Yaskawa INFORM job: X2_101(P)NEWKM.JBI

/JOB
//NAME X2_101(P)NEWKM
//POS
///NPOS 465,465,465,24,0,0
///TOOL 0
///POSTYPE PULSE
///PULSE
C00000=3858,45070,-46943,-23358,97175,-79306
C00001=-126163,171030,121698,-25332,17066,-72423
///LIMIT ON
C00002=-15532,205449,169164,0,-1122,-37
C00003=-2035,205524,169313,0,-1142,-38
///LIMIT OFF
C00004=-24876,216658,221537,-34735,41227,28422
C00005=-32534,213651,221430,-43713,46730,30831
C00006=-90550,189136,203825,-30202,58765,18284
C00007=-119585,140470,218769,-27614,53519,-2911
C00008=-120519,138494,231532,-24554,52332,-6677
C00009=-121361,123084,224135,-22504,53325,-9347
C00010=-121726,115435,217146,-22627,53645,-9461
C00011=-121876,112275,214159,-22659,53833,-9521
C00012=-121870,108701,209945,-22450,54535,-9681
C00013=-121878,109205,210521,-22481,54446,-9661
C00014=-121910,109175,212145,-22779,53504,-9448
C00015=-121878,109205,210521,-22481,54446,-9661
C00016=-121362,120230,220888,-22358,53819,-9461
C00017=-121399,123144,224213,26030,40987,26163
C00018=-121766,115498,217228,25645,41349,26232
C00019=-121913,110359,211916,25262,41930,26397
C00020=-121910,108768,210034,25105,42240,26494
C00021=-121911,109318,210663,25153,42145,26465
C00022=-121945,109286,212284,25618,41227,26168
C00023=-121911,109318,210663,25153,42145,26465
C00024=-121395,120334,221016,25773,41460,26319
C00025=-121834,122785,223550,29969,46824,26161
C00026=-121859,115436,217233,29902,46923,26193
C00027=-121866,110818,212669,29698,47304,26325
C00028=-121863,108844,210335,29512,47673,26452
C00029=-121935,109447,211025,29521,47579,26410
C00030=-121969,109405,212635,29961,46698,26100
C00031=-121935,109447,211025,29521,47579,26410
C00032=-121897,120013,220389,29693,47285,26314
C00033=-121710,149750,244683,33916,46787,25442
C00034=-122130,167084,227684,35838,62010,28886
C00035=-121679,161325,224182,36290,61247,28722
C00036=-121494,157054,220841,36419,61089,28713
C00037=-121492,155796,219623,36386,61172,28744
C00038=-121498,156274,220057,36390,61156,28737
C00039=-121513,157313,222807,36761,60220,28378
C00040=-121498,156274,220057,36390,61156,28737
C00041=-122131,164491,225278,35793,62131,28930
C00042=-121153,166943,227356,19598,60055,30811
C00043=-121390,161131,223816,19656,59323,30620
C00044=-121486,157179,220857,19658,59138,30564
C00045=-121483,155572,219231,19626,59303,30596
C00046=-121495,156085,219721,19629,59269,30586
C00047=-121510,157133,222481,19854,58176,30378
C00048=-121495,156085,219721,19629,59269,30586
C00049=-121161,164380,224998,19569,60183,30833
C00050=-134270,166899,227330,-30052,67117,-21044
C00051=-134672,161022,223642,-30400,66383,-20931
C00052=-134827,157380,220874,-30511,66205,-20916
C00053=-134816,155436,218995,-30471,66344,-20953
C00054=-134842,155930,219452,-30490,66315,-20951
C00055=-135058,156963,222167,-30845,65285,-20702
C00056=-134842,155930,219452,-30490,66315,-20951
C00057=-134278,164319,224942,-30027,67241,-21080
C00058=-134522,188621,240209,-29351,55882,-39556
C00059=-134281,187845,227413,-27061,47780,-60505
C00060=-134637,183113,225522,-27632,46565,-60252
C00061=-134774,179835,223566,-27858,46107,-60152
C00062=-134763,178280,222255,-27854,46115,-60152
C00063=-134775,178711,222615,-27856,46112,-60156
C00064=-134965,180234,225747,-28400,45052,-59871
C00065=-134775,178711,222615,-27856,46112,-60156
C00066=-134277,185474,225522,-27083,47733,-60488
C00067=-128103,202093,243005,-900,47088,-2105
C00068=-121693,187846,227414,25459,51264,56132
C00069=-121495,183214,225706,25955,50017,55854
C00070=-121414,180043,223882,26152,49543,55743
C00071=-121411,178420,222512,26150,49549,55748
C00072=-121403,178860,222872,26150,49552,55751
C00073=-121416,180408,226053,26590,48508,55442
C00074=-121403,178860,222872,26150,49552,55751
C00075=-121682,185481,225516,25477,51219,56123
C00076=-121689,188183,227953,25513,51119,56094
C00077=-121490,183546,226247,26015,49869,55812
C00078=-121408,180079,224179,26215,49393,55704
C00079=-121407,178755,223064,26213,49397,55705
C00080=-121411,179182,223381,26203,49420,55711
C00081=-121423,180718,226547,26645,48380,55401
C00082=-121411,179182,223381,26203,49420,55711
C00083=-121690,185807,226020,25524,51091,56086
C00084=-123779,190470,236318,58172,45370,-30510
C00085=-122063,184657,229672,57761,45274,-29622
C00086=-121391,180820,225681,57548,45265,-29244
C00087=-121389,179381,224477,57547,45264,-29243
C00088=-121377,179861,224816,57519,45280,-29221
C00089=-121365,178277,221590,56564,45934,-28599
C00090=-121377,179861,224816,57519,45280,-29221
C00091=-121233,179889,223673,56966,45622,-28813
C00092=-120840,179898,223685,57074,45455,-28743
C00093=-121856,179870,223641,56791,45888,-28921
C00094=-124230,188212,233297,57460,45939,-30216
C00095=-135456,214682,237929,8760,44354,-9002
C00096=-135014,207234,230989,8630,44755,-8792
C00097=-134830,202547,226948,8592,44816,-8716
C00098=-134825,201671,226346,8603,44738,-8721
C00099=-134842,202253,226813,8604,44750,-8727
C00100=-134670,200231,223307,8417,45842,-8557
C00101=-134842,202253,226813,8604,44750,-8727
C00102=-135456,212819,236850,8805,44063,-9030
C00103=-144745,210021,243410,8185,41273,-14023
C00104=-162917,179999,233290,6575,38143,-23957
C00105=-161998,172707,226275,6517,38664,-23607
C00106=-162887,167099,219775,6342,39818,-23812
C00107=-162887,165781,218634,6340,39844,-23811
C00108=-162887,166055,218871,6340,39839,-23811
C00109=-162343,164612,215992,6206,40837,-23555
C00110=-162887,166055,218871,6340,39839,-23811
C00111=-162962,177992,231819,6593,38021,-23983
C00112=-147831,180663,236712,-46705,20975,10626
C00113=-148148,173122,227595,-43517,22125,9005
C00114=-148274,168937,222870,-42234,22650,8350
C00115=-148281,167110,221344,-42230,22650,8346
C00116=-148302,167857,221980,-42238,22637,8344
C00117=-147925,166248,218822,-40599,23599,7656
C00118=-148302,167857,221980,-42238,22637,8344
C00119=-147863,178628,235160,-46872,20902,10696
C00120=-134462,161839,227541,-33778,50638,-10353
C00121=-128292,130528,217892,-31335,63768,-21724
C00122=-129684,119449,220047,-34318,57761,-20007
C00123=-130320,112373,214177,-34735,57677,-20053
C00124=-130456,109465,211770,-34840,57652,-20062
C00125=-133214,109388,211257,-36497,57589,-20371
C00126=-136667,109271,210511,-38562,57521,-20784
C00127=-139224,109161,209855,-40060,57485,-21111
C00128=-138850,112080,212320,-39829,57519,-21074
C00129=-138002,119182,218308,-39302,57595,-20992
C00130=-116829,118715,218073,25020,47867,39145
C00131=-117081,112091,213071,24998,47591,39033
C00132=-116945,109370,210997,25124,47467,39017
C00133=-125403,109328,210939,20229,48081,38115
C00134=-125748,112035,212901,19975,48276,38114
C00135=-125224,118667,217955,20186,48522,38233
C00136=-124121,120753,219622,35413,60229,26204
C00137=-123486,114299,214861,35950,59841,26140
C00138=-122342,111487,212696,36731,59624,26198
C00139=-123646,102227,205116,46204,63991,23691
C00140=-125197,104926,207303,45145,64225,23601
C00141=-126541,111461,212474,44185,64527,23570
C00142=-123354,156374,234537,36141,60524,36841
C00143=-123006,163587,222304,33363,70023,40058
C00144=-122562,159556,221336,33872,68682,39742
C00145=-122328,157903,220938,34117,68123,39618
C00146=-120667,157882,220896,34940,67759,39903
C00147=-118950,157779,220838,35793,67346,40185
C00148=-123086,151768,218649,44650,69367,37665
C00149=-123645,153585,219325,44221,69895,37762
C00150=-124560,157673,220588,43425,71117,38069
C00151=-118179,162280,221931,19519,66647,42953
C00152=-118374,158121,220823,19639,65298,42675
C00153=-118267,155527,219476,19766,64809,42612
C00154=-124138,155466,219359,17061,65585,41471
C00155=-124017,158021,220644,17053,66071,41570
C00156=-123705,162202,221801,17023,67409,41838
C00157=-131226,163758,224551,-30632,74582,-25473
C00158=-131671,158900,222412,-31029,73469,-25265
C00159=-131767,156865,221384,-31140,73093,-25182
C00160=-137554,155593,218490,-34050,72807,-26431
C00161=-137282,157641,219617,-33852,73169,-26479
C00162=-136745,162505,221837,-33401,74244,-26683
C00163=-132458,177728,230704,-28826,51363,-58996
C00164=-131589,185090,225420,-26277,57937,-60697
C00165=-131989,181524,225146,-26843,56352,-60401
C00166=-132129,179690,224573,-27052,55792,-60292
C00167=-137018,178141,221655,-27936,55567,-61763
C00168=-136911,179846,222046,-27715,56157,-61897
C00169=-136440,196977,232068,-26852,58624,-62420
C00170=-123981,183157,222393,21512,66418,58052
C00171=-123825,180405,223212,21872,64600,57740
C00172=-123515,178835,223292,22117,63748,57656
C00173=-118554,178759,223273,23717,62772,58838
C00174=-118823,180539,223431,23475,63574,58935
C00175=-119074,183322,222662,23052,65379,59248
C00176=-122702,184077,222510,27150,66928,58165
C00177=-122303,181421,223407,27656,65122,57824
C00178=-121939,179837,223488,27962,64268,57706
C00179=-119147,179825,223466,28889,63614,58349
C00180=-122880,176137,223692,38896,64069,56161
C00181=-123433,177900,223899,38463,64850,56297
C00182=-124245,180658,223301,37680,66520,56676
C00183=-126373,202040,241637,26852,43466,21020
C00184=-128666,178893,235276,24840,16714,-14065
C00185=-128229,171381,226060,22241,18307,-12727
C00186=-128063,167759,221784,21279,19001,-12231
C00187=-126454,168065,222273,20329,18606,-11329
C00188=-113498,168020,221950,9782,17256,-2783
C00189=-116924,165235,218756,37372,21894,-17093
C00190=-117333,168644,222995,38850,21324,-17919
C00191=-117978,176136,232334,42331,20047,-19764
C00192=-122460,189534,236128,2418,24460,-9718
C00193=-126271,180528,223816,-31550,27550,-1309
C00194=-126367,172058,213874,-29849,29054,-2198
C00195=-127090,167664,208219,-28567,29945,-3048
C00196=-142506,160672,196064,-19689,30087,-11601
C00197=-142606,164949,201311,-20262,29094,-11331
C00198=-142831,174249,212461,-21540,27099,-10741
C00199=-90550,189136,203825,-30202,58765,18284
C00200=-32534,213651,221430,-43713,46730,30831
///LIMIT ON
C00201=-2035,205524,169313,0,-1142,-38
///LIMIT OFF
C00202=110357,194361,192639,11084,17793,24068
C00203=114624,170501,213981,27000,30394,20280
C00204=117760,152303,229663,38696,39653,17494
C00205=136745,136971,237540,47053,40245,16937
C00206=147677,120644,222935,49307,45765,18910
C00207=147943,109722,211385,48401,46737,19631
C00208=147915,107740,209041,48089,47029,19824
C00209=147921,108247,209621,48160,46963,19780
C00210=148534,108214,211137,49208,46239,19387
C00211=147921,108247,209621,48160,46963,19780
C00212=146752,119366,220398,48075,46495,19266
C00213=146769,122228,223642,-12245,42312,-23405
C00214=147600,114525,216379,-11673,42843,-23379
C00215=143912,110143,217361,-5106,40312,-21729
C00216=143912,106051,212649,-5023,41107,-21780
C00217=143912,106490,213159,-5032,41020,-21775
C00218=144459,106367,214517,-4806,40132,-21665
C00219=143912,108428,215397,-5071,40640,-21751
C00220=146723,119408,220432,-12150,42825,-23484
C00221=143045,138896,235476,-13742,43230,-24222
C00222=120960,164034,232760,-20897,55487,-30119
C00223=121057,160229,229930,-20909,55300,-30059
C00224=121055,158546,228333,-20881,55408,-30082
C00225=121067,159042,228799,-20882,55381,-30074
C00226=121067,159823,231250,-21156,54345,-29857
C00227=121067,159042,228799,-20882,55381,-30074
C00228=120732,167440,234058,-20772,56349,-30345
C00229=148415,169733,235789,37593,61151,22296
C00230=149007,163695,231894,38120,60456,22164
C00231=149231,159863,228946,38284,60282,22149
C00232=149211,158151,227325,38234,60380,22184
C00233=149239,158627,227750,38254,60361,22183
C00234=149676,159369,230053,38836,59445,21914
C00235=149239,158627,227750,38254,60361,22183
C00236=148408,167213,233502,37553,61243,22331
C00237=120948,174757,250553,37714,32624,49250
C00238=118901,165188,232218,31966,38533,51583
C00239=120946,159930,222884,30547,40745,53182
C00240=121038,156296,220141,30673,40571,53142
C00241=121036,154340,218237,30574,40715,53200
C00242=121048,154616,218515,30593,40687,53192
C00243=121049,155465,220596,31099,39958,52886
C00244=121048,154822,218707,30600,40677,53188
C00245=120729,163160,224069,29968,41598,53447
C00246=121377,165750,226457,-30289,41550,-53313
C00247=121143,159913,222862,-30795,40818,-53099
C00248=121047,156279,220118,-30922,40645,-53059
C00249=121045,154323,218215,-30823,40788,-53119
C00250=121036,154817,218686,-30845,40755,-53109
C00251=121036,155874,221461,-31554,39751,-52691
C00252=121036,154817,218686,-30845,40755,-53109
C00253=121366,163152,224045,-30207,41677,-53367
C00254=121366,163152,224045,-30207,41677,-53367
C00255=121483,199612,234227,-6189,47888,801
C00256=116205,204502,245408,11942,36344,-5913
C00257=116205,198287,241356,12142,35658,-6024
C00258=115285,196386,239785,12255,35742,-6372
C00259=115285,194113,238215,12313,35542,-6405
C00260=115285,196386,239785,12255,35742,-6372
C00261=115348,194991,237157,11988,36617,-6206
C00262=115285,196386,239785,12255,35742,-6372
C00263=123104,195479,239507,19665,35466,-6181
C00264=123104,195479,239507,19665,35466,-6181
C00265=123104,193192,237914,19758,35282,-6230
C00266=123104,195479,239507,19665,35466,-6181
C00267=123076,194119,236930,19261,36311,-5967
C00268=123104,195479,239507,19665,35466,-6181
C00269=121128,212741,249815,-1743,43167,1820
C00270=122107,209686,246756,-2334,35321,2429
C00271=122102,206275,244139,-2341,35179,2433
C00272=122102,203894,242650,-2356,34872,2441
C00273=122102,204632,243115,-2351,34965,2438
C00274=122089,203132,240589,-2306,35750,2407
C00275=122102,206496,244275,-2336,35209,2431
C00276=106576,204382,240236,-11557,35635,-12
C00277=105844,202338,238595,-11416,35522,-303
C00278=105844,200288,237272,-11482,35287,-265
C00279=105844,200808,237609,-11466,35345,-274
C00280=105986,199498,235274,-11288,36108,-332
C00281=106675,205315,241966,-11744,35073,120
C00282=121297,207453,245813,-14870,35545,6164
C00283=121834,203391,244226,-16112,31944,7027
C00284=106221,199743,239162,-19916,31296,2840
C00285=113509,210579,250034,-22345,31553,6212
C00286=137477,186722,245503,32144,20066,-8132
C00287=144465,175669,236908,30012,18300,-5031
C00288=139549,172315,235287,31351,18759,-7203
C00289=137345,164078,227518,10851,18120,-89
C00290=146058,157132,216606,32577,20921,-6799
C00291=140284,173520,236299,40392,19304,-12229
C00292=141359,173291,233520,11184,20569,1731
C00293=118409,183246,223281,22704,61297,57282
C00294=118581,179790,223172,23116,59682,56982
C00295=119080,177311,221631,23320,59284,57040
C00296=121941,178499,224734,27845,56338,58798
C00297=123595,179764,223148,24469,58676,58234
C00298=123340,183247,223305,24003,60279,58531
C00299=123969,187046,227095,-21794,65540,-58072
C00300=123769,179484,222767,-22062,64364,-57894
C00301=123576,177800,222588,-22257,63628,-57801
C00302=118799,177973,222710,-23788,62722,-58944
C00303=118761,179531,222831,-23662,63378,-59098
C00304=119022,182337,222102,-23232,65173,-59409
C00305=118548,185960,240006,-23112,60518,-52609
C00306=118308,157164,220237,-19921,65161,-42814
C00307=118476,159354,225951,-20677,60172,-41891
C00308=123703,159378,225931,-18342,60853,-40897
C00309=124532,167340,231429,-17858,61624,-40849
C00310=131317,177717,239716,826,64580,-18015
C00311=127714,174798,240675,21893,68906,13109
C00312=128493,175754,243778,32993,66237,18094
C00313=129602,162263,233964,31751,67819,21399
C00314=133248,162950,235869,37514,65238,22588
C00315=131009,170167,241494,36207,65881,22354
C00316=129314,152311,241224,32836,60701,20495
C00317=134262,125348,219975,36015,59621,20953
C00318=135447,125082,223354,38338,54808,19572
C00319=142546,124299,220540,42255,55214,20638
C00320=139661,130867,226583,40618,55342,20260
C00321=128999,132996,229263,10730,53492,-5640
C00322=116671,118195,219736,-25901,46707,-38928
C00323=118115,111302,212748,-24760,47506,-38978
C00324=115332,106344,206919,-23218,48620,-39011
C00325=123639,106372,207077,-18510,49117,-38052
C00326=123644,119783,222350,-19919,44975,-37125
C00327=114229,133215,224760,-34569,55636,-15897
C00328=115215,137513,213650,-31198,63454,-18326
C00329=115698,129470,194907,-29425,69976,-20075
C00330=106762,152299,200628,-28970,57173,-24551
C00331=110317,154116,190151,-51141,5677,-13903
C00332=107071,171086,183471,-26129,-3539,-25752
C00333=106762,173596,155880,-23749,-4416,-26879
C00334=27327,173596,155880,-23749,-4416,-26879
C00335=61821,209309,227101,13653,32656,17858
C00336=117760,152303,229663,38696,39653,17494
C00337=136745,136971,237540,47053,40245,16937
C00338=146994,113665,215692,48512,45897,19228
C00339=147943,109722,211385,48401,46737,19631
C00340=147915,107740,209041,48089,47029,19824
C00341=147921,108247,209621,48160,46963,19780
C00342=148534,108214,211137,49208,46239,19387
C00343=147921,108247,209621,48160,46963,19780
C00344=146752,119366,220398,48075,46495,19266
C00345=146769,122228,223642,-12245,42312,-23405
C00346=147600,114525,216379,-11673,42843,-23379
C00347=150410,110151,217690,-10757,39930,-22674
C00348=147891,107738,209025,-11299,43871,-23478
C00349=153573,108674,222079,-9620,36586,-21959
C00350=148504,108258,211178,-11182,42854,-23269
C00351=153573,108674,222079,-9620,36586,-21959
C00352=146723,119408,220432,-12150,42825,-23484
C00353=145733,131948,231566,-12791,42388,-23541
C00354=120722,165761,226456,-19970,59936,-31049
C00355=120948,159926,222866,-20032,59223,-30862
C00356=121040,156088,219926,-20029,59083,-30814
C00357=121038,154338,218222,-19999,59222,-30841
C00358=121049,154854,218719,-20002,59186,-30831
C00359=121049,155913,221496,-20240,58090,-30621
C00360=121049,154854,218719,-20002,59186,-30831
C00361=120732,163185,224070,-19939,60073,-31072
C00362=147021,165785,226508,35831,64459,23179
C00363=147568,159794,222565,36267,63796,23080
C00364=147776,155921,219507,36395,63658,23083
C00365=147758,154144,217781,36345,63784,23124
C00366=147784,154635,218233,36365,63757,23122
C00367=148179,155632,220846,36870,62776,22859
C00368=147784,154635,218233,36365,63757,23122
C00369=147016,163193,224095,35787,64586,23223
C00370=120935,171934,242189,34504,35645,50983
C00371=120720,165768,226479,30046,41476,53396
C00372=120946,159930,222884,30547,40745,53182
C00373=121038,156296,220141,30673,40571,53142
C00374=121036,154340,218237,30574,40715,53200
C00375=121048,154616,218515,30593,40687,53192
C00376=121049,155465,220596,31099,39958,52886
C00377=121048,154822,218707,30600,40677,53188
C00378=120729,163160,224069,29968,41598,53447
C00379=121377,165750,226457,-30289,41550,-53313
C00380=121143,159913,222862,-30795,40818,-53099
C00381=121047,156279,220118,-30922,40645,-53059
C00382=121045,154323,218215,-30823,40788,-53119
C00383=121036,154817,218686,-30845,40755,-53109
C00384=121036,155874,221461,-31554,39751,-52691
C00385=121036,154817,218686,-30845,40755,-53109
C00386=121366,163152,224045,-30207,41677,-53367
C00387=137298,197580,228407,-4602,50872,8306
C00388=150104,186063,215083,4172,47395,10089
C00389=151037,187915,222611,5560,37459,9696
C00390=151037,185231,220636,5579,37292,9686
C00391=151037,186381,221487,5571,37359,9691
C00392=150722,184726,218590,5524,38303,9628
C00393=151037,186381,221487,5571,37359,9691
C00394=146916,195279,232433,6810,35442,7817
C00395=137844,201998,246759,9498,27003,3396
C00396=137686,197394,242433,9461,27307,3368
C00397=137686,195263,240973,9523,27113,3337
C00398=137686,196472,241804,9489,27221,3355
C00399=137493,195182,239322,9290,28089,3401
C00400=137686,196472,241804,9489,27221,3355
C00401=137872,200789,246191,9576,26732,3366
C00402=125774,205155,244676,-1779,39656,5291
C00403=112923,203838,248508,-13462,25066,7526
C00404=112273,198134,243408,-13075,25198,7148
C00405=112273,195800,241814,-13181,24982,7201
C00406=112273,196433,242252,-13153,25040,7187
C00407=112372,195114,239703,-12779,25919,7028
C00408=112273,198506,243659,-13056,25235,7140
C00409=116013,198964,244548,-14816,25354,9073
C00410=116342,198570,244149,-14930,25435,9223
C00411=116342,196143,242500,-15057,25209,9285
C00412=116342,196705,242885,-15029,25259,9270
C00413=116387,195582,240705,-14639,26004,9089
C00414=116342,197910,243703,-14967,25370,9239
C00415=117942,195646,241316,-14532,25786,9480
C00416=100647,189294,231884,-21448,26183,5644
C00417=105174,198018,242573,-25014,25112,8670
C00418=138600,188940,247456,26519,19021,-5159
C00419=137571,174455,238189,28708,17651,-6518
C00420=137161,164520,226883,26329,19378,-5524
C00421=155042,153638,205005,15246,25339,2538
C00422=152712,160990,215450,17982,23102,538
C00423=143867,184578,245341,28376,18738,-7025
C00424=118409,183246,223281,22704,61297,57282
C00425=118581,179790,223172,23116,59682,56982
C00426=118693,177304,221659,23221,59339,56941
C00427=123485,177367,221685,24518,58397,58134
C00428=123595,179764,223148,24469,58676,58234
C00429=123340,183247,223305,24003,60279,58531
C00430=123938,190075,227776,-21625,66593,-58285
C00431=123769,179484,222767,-22062,64364,-57894
C00432=123184,178126,222935,-22395,63511,-57887
C00433=118491,177814,222796,-23918,62536,-58992
C00434=118761,179531,222831,-23662,63378,-59098
C00435=119022,182337,222102,-23232,65173,-59409
C00436=122719,191364,242917,-21569,61694,-52463
C00437=118308,157164,220237,-19921,65161,-42814
C00438=118111,154516,218858,-20091,64650,-42768
C00439=123565,154529,218888,-17585,65335,-41706
C00440=123968,157132,220198,-17330,65894,-41703
C00441=123666,171172,229916,-17315,67038,-41943
C00442=144355,163571,225284,37353,71372,27423
C00443=145029,158578,222871,37922,70344,27214
C00444=145301,156779,221933,38139,70000,27151
C00445=150377,154595,216968,40372,70234,28530
C00446=150395,156248,217650,40288,70560,28668
C00447=149652,161243,220185,39700,71542,28858
C00448=132795,148549,237387,35039,60818,21489
C00449=129694,120788,221943,34103,57517,19821
C00450=131382,111553,213551,35044,57698,20084
C00451=141801,108057,208206,41145,57678,21431
C00452=149498,107271,204816,45301,57831,22696
C00453=138916,111308,211941,39557,57554,20977
C00454=138073,118434,217968,39036,57618,20892
C00455=116671,118195,219736,-25901,46707,-38928
C00456=118115,111302,212748,-24760,47506,-38978
C00457=116900,108123,210017,-25446,47458,-39118
C00458=125154,108371,210177,-20660,48073,-38243
C00459=125733,111262,212625,-20332,48091,-38177
C00460=125221,117920,217723,-20539,48325,-38292
C00461=126776,138177,229575,-26069,55844,-18031
C00462=78165,188060,235135,7900,30611,9082
C00463=59194,210722,234815,16854,29215,15555
C00464=-5072,204191,177105,2520,2910,2072
BC00000=46343,515539,1075137
BC00001=134211,257442,1075137
BC00002=1577,514581,1075193
///LIMIT ON
BC00003=1577,-59411,1075193
BC00004=21651,-83121,1075193
BC00005=24420,-86391,1075193
BC00006=182796,-159531,881707
BC00007=261191,-81513,996983
BC00008=265032,-63260,961437
BC00009=267226,-52830,941125
BC00010=267226,-52830,941125
BC00011=267226,-52830,941125
BC00012=267226,-52830,941125
BC00013=267226,-52830,941125
BC00014=267226,-52830,941125
BC00015=267226,-52830,941125
BC00016=267226,-52830,941125
BC00017=280671,-69653,979309
BC00018=280671,-69653,979309
BC00019=280671,-69653,979309
BC00020=280671,-69653,979309
BC00021=280671,-69653,979309
BC00022=280671,-69653,979309
BC00023=280671,-69653,979309
BC00024=280671,-69653,979309
BC00025=340059,-63189,958778
BC00026=340059,-63189,958778
BC00027=340059,-63189,958778
BC00028=340059,-63189,958778
BC00029=340059,-63189,958778
BC00030=340059,-63189,958778
BC00031=340059,-63189,958778
BC00032=340059,-63189,958778
BC00033=335398,-76723,919166
BC00034=322582,-113941,810232
BC00035=322582,-113941,810232
BC00036=322582,-113941,810232
BC00037=322582,-113941,810232
BC00038=322582,-113941,810232
BC00039=322582,-113941,810232
BC00040=322582,-113941,810232
BC00041=322582,-113941,810232
BC00042=280667,-107560,836160
BC00043=280667,-107560,836160
BC00044=280667,-107560,836160
BC00045=280667,-107560,836160
BC00046=280667,-107560,836160
BC00047=280667,-107560,836160
BC00048=280667,-107560,836160
BC00049=280667,-107560,836160
BC00050=310567,-93619,803899
BC00051=310567,-93619,803899
BC00052=310567,-93619,803899
BC00053=310567,-93619,803899
BC00054=310567,-93619,803899
BC00055=310567,-93619,803899
BC00056=310567,-93619,803899
BC00057=310567,-93619,803899
BC00058=310965,-106510,799405
BC00059=311390,-120260,794612
BC00060=311390,-120260,794612
BC00061=311390,-120260,794612
BC00062=311390,-120260,794612
BC00063=311390,-120260,794612
BC00064=311390,-120260,794612
BC00065=311390,-120260,794612
BC00066=311390,-120260,794612
BC00067=292086,-121797,794251
BC00068=272781,-123335,793890
BC00069=272781,-123335,793890
BC00070=272781,-123335,793889
BC00071=272781,-123335,793890
BC00072=272781,-123335,793890
BC00073=272781,-123335,793890
BC00074=272781,-123335,793890
BC00075=272781,-123335,793890
BC00076=341329,-123426,794084
BC00077=341329,-123426,794084
BC00078=341329,-123426,794084
BC00079=341329,-123426,794084
BC00080=341329,-123426,794084
BC00081=341329,-123426,794084
BC00082=341329,-123426,794084
BC00083=341329,-123426,794084
BC00084=311173,-145946,723752
BC00085=311173,-145946,723752
BC00086=311173,-145946,723752
BC00087=311173,-145946,723752
BC00088=311173,-145946,723752
BC00089=311173,-145946,723752
BC00090=311173,-145946,723752
BC00091=311173,-145946,723752
BC00092=311173,-145946,723752
BC00093=311173,-145946,723752
BC00094=311173,-145946,723752
BC00095=368417,-159833,659013
BC00096=368417,-159833,659013
BC00097=368417,-159833,659013
BC00098=368417,-159833,659013
BC00099=368417,-159833,659013
BC00100=368417,-159833,659013
BC00101=368417,-159833,659013
BC00102=368417,-159833,659013
BC00103=371175,-130977,746316
BC00104=376801,-72111,924416
BC00105=376801,-72111,924416
BC00106=376801,-72111,924416
BC00107=376801,-72111,924416
BC00108=376801,-72111,924416
BC00109=376801,-72111,924414
BC00110=376801,-72111,924416
BC00111=376801,-72111,924416
BC00112=341502,-110623,881707
BC00113=341502,-110623,881707
BC00114=341502,-110623,881707
BC00115=341502,-110623,881707
BC00116=341502,-110623,881707
BC00117=341502,-110623,881707
BC00118=341502,-110623,881707
BC00119=341502,-110623,881707
BC00120=317229,-102231,901443
BC00121=301231,-72103,952987
BC00122=300570,-48582,912240
BC00123=300570,-48582,912240
BC00124=300570,-48582,912238
BC00125=300570,-48582,912240
BC00126=300570,-48582,912240
BC00127=300570,-48582,912240
BC00128=300570,-48582,912240
BC00129=300570,-48582,912240
BC00130=280392,-58723,951442
BC00131=280392,-58723,951442
BC00132=280392,-58723,951442
BC00133=280392,-58723,951442
BC00134=280392,-58723,951442
BC00135=280392,-58723,951442
BC00136=316381,-56573,892692
BC00137=316381,-56573,892692
BC00138=316381,-56573,892692
BC00139=316381,-56573,892692
BC00140=316381,-56573,892692
BC00141=316381,-56573,892692
BC00142=316378,-102850,892874
BC00143=316296,-103943,772800
BC00144=316296,-103943,772800
BC00145=316296,-103943,772800
BC00146=316296,-103943,772800
BC00147=316296,-103943,772800
BC00148=316296,-103943,772800
BC00149=316296,-103943,772800
BC00150=316296,-103943,772800
BC00151=280455,-96630,809993
BC00152=280455,-96630,809993
BC00153=280455,-96630,809993
BC00154=280455,-96630,809993
BC00155=280455,-96630,809993
BC00156=280455,-96630,809993
BC00157=313485,-85360,768647
BC00158=313485,-85360,768647
BC00159=313485,-85360,768647
BC00160=313485,-85360,768647
BC00161=313485,-85360,768647
BC00162=313485,-85360,768647
BC00163=312825,-103474,920081
BC00164=312211,-104211,778577
BC00165=312211,-104211,778577
BC00166=312212,-104211,778575
BC00167=312212,-104211,778575
BC00168=312211,-104211,778577
BC00169=312211,-104211,778577
BC00170=271148,-98769,766614
BC00171=271148,-98769,766614
BC00172=271148,-98769,766614
BC00173=271148,-98769,766614
BC00174=271148,-98769,766614
BC00175=271148,-98769,766614
BC00176=325606,-102154,751502
BC00177=325606,-102154,751502
BC00178=325606,-102154,751502
BC00179=325606,-102154,751502
BC00180=325606,-102154,751502
BC00181=325606,-102154,751502
BC00182=325606,-102154,751502
BC00183=333034,-134164,767871
BC00184=339129,-149656,848222
BC00185=339129,-149656,848222
BC00186=339128,-149655,848221
BC00187=339129,-149656,848222
BC00188=339129,-149656,848222
BC00189=339129,-149656,848222
BC00190=339129,-149656,848222
BC00191=339129,-149656,848222
BC00192=327972,-150195,844855
BC00193=317352,-148908,839217
BC00194=317352,-148908,839217
BC00195=317352,-148908,839217
BC00196=317352,-148908,839217
BC00197=317352,-148908,839217
BC00198=317352,-148908,839217
BC00199=182796,-159531,881707
BC00200=24420,-86391,1075193
BC00201=1577,-59411,1075193
///LIMIT OFF
BC00202=66886,568997,1042628
BC00203=92444,428784,1010343
BC00204=92897,349346,986620
BC00205=164885,323227,963040
BC00206=185515,310988,951990
BC00207=185515,310988,951990
BC00208=185515,310988,951990
BC00209=185515,310988,951990
BC00210=185515,310988,951990
BC00211=185515,310988,951990
BC00212=185515,310988,951990
BC00213=189482,318421,980677
BC00214=189482,318421,980677
BC00215=189482,306857,980677
BC00216=189482,306857,980677
BC00217=189482,306857,980677
BC00218=189482,306857,980677
BC00219=189482,306857,980677
BC00220=189482,318421,980677
BC00221=182754,323413,960497
BC00222=141913,353717,838001
BC00223=141913,353717,838001
BC00224=141913,353717,838001
BC00225=141913,353717,838001
BC00226=141913,353717,838001
BC00227=141913,353717,838001
BC00228=141913,353717,838001
BC00229=207263,329283,804361
BC00230=207263,329283,804361
BC00231=207263,329283,804361
BC00232=207263,329283,804361
BC00233=207263,329283,804361
BC00234=207263,329283,804361
BC00235=207263,329283,804361
BC00236=207263,329283,804361
BC00237=131545,342192,928572
BC00238=131545,342192,928572
BC00239=131545,352945,928572
BC00240=131545,352945,928572
BC00241=131545,352945,928572
BC00242=131545,352945,928572
BC00243=131546,352945,928571
BC00244=131545,352945,928572
BC00245=131545,352945,928572
BC00246=134650,353410,929381
BC00247=134650,353410,929381
BC00248=134650,353410,929381
BC00249=134650,353410,929381
BC00250=134650,353410,929381
BC00251=134650,353410,929381
BC00252=134650,353410,929381
BC00253=134650,353410,929381
BC00254=134650,353410,929381
BC00255=134373,390505,753296
BC00256=93548,390505,753296
BC00257=93548,390505,753296
BC00258=93548,390505,753296
BC00259=93548,390505,753296
BC00260=93548,390505,753296
BC00261=93548,390505,753296
BC00262=93548,390505,753296
BC00263=93548,390505,753296
BC00264=93548,390505,753296
BC00265=93548,390505,753296
BC00266=93548,390505,753296
BC00267=93548,390505,753296
BC00268=93548,390505,753296
BC00269=168621,382981,746953
BC00270=168621,382981,746953
BC00271=168621,382981,746953
BC00272=168621,382981,746953
BC00273=168621,382981,746953
BC00274=168621,382981,746953
BC00275=168621,382981,746953
BC00276=147987,382981,746953
BC00277=147987,382981,746953
BC00278=147987,382981,746953
BC00279=147987,382981,746953
BC00280=147987,382981,746953
BC00281=147987,382981,746953
BC00282=147987,382981,746953
BC00283=148413,382917,748107
BC00284=148720,382872,748941
BC00285=148720,382872,748941
BC00286=202687,374937,895402
BC00287=202687,374937,895402
BC00288=181755,375248,897598
BC00289=159634,375248,897598
BC00290=159830,375278,897817
BC00291=159830,375278,897817
BC00292=181599,378656,922199
BC00293=133265,363347,778304
BC00294=133265,363347,778304
BC00295=133265,363348,778302
BC00296=133265,363347,778303
BC00297=133265,363347,778304
BC00298=133265,363347,778304
BC00299=146867,355192,768709
BC00300=133835,355192,768709
BC00301=133835,355192,768709
BC00302=133835,355192,768709
BC00303=133835,355192,768709
BC00304=133835,355192,768709
BC00305=137056,354441,784011
BC00306=142942,353070,811970
BC00307=142942,353070,811970
BC00308=142942,353070,811970
BC00309=142942,353070,811970
BC00310=165851,345786,796984
BC00311=162229,334955,774700
BC00312=164558,332161,768952
BC00313=169097,331686,770079
BC00314=169097,331686,770079
BC00315=169097,331686,770079
BC00316=172928,318668,849125
BC00317=172716,318424,871943
BC00318=172716,318424,871943
BC00319=172716,318424,871943
BC00320=172716,318424,871943
BC00321=159709,316953,907603
BC00322=143169,315083,952947
BC00323=143169,315083,952947
BC00324=143169,315083,952947
BC00325=143169,315083,952947
BC00326=143169,315083,952947
BC00327=119317,333024,923162
BC00328=123697,333024,923162
BC00329=132263,359008,1050367
BC00330=116798,380944,1050367
BC00331=119098,435388,1050366
BC00332=102300,494697,1050367
BC00333=98226,585882,1050367
BC00334=13715,585882,1050367
BC00335=124194,427082,1056800
BC00336=295181,349346,986620
BC00337=336555,323227,963040
BC00338=354347,311995,952900
BC00339=355943,310988,951990
BC00340=355943,310988,951990
BC00341=355943,310988,951990
BC00342=355943,310988,951990
BC00343=355943,310988,951990
BC00344=355943,310988,951990
BC00345=359910,318421,980677
BC00346=359910,318421,980677
BC00347=359910,306857,980677
BC00348=359910,318421,980677
BC00349=359910,294465,980677
BC00350=359910,318421,980677
BC00351=359910,294465,980677
BC00352=359910,318421,980677
BC00353=359910,318421,980677
BC00354=312341,364470,838001
BC00355=312341,364470,838001
BC00356=312341,364470,838001
BC00357=312341,364470,838001
BC00358=312341,364470,838001
BC00359=312341,364470,838001
BC00360=312341,364470,838001
BC00361=312341,364470,838001
BC00362=377691,340036,804361
BC00363=377691,340036,804361
BC00364=377691,340036,804361
BC00365=377691,340036,804361
BC00366=377691,340036,804361
BC00367=377691,340036,804361
BC00368=377691,340036,804361
BC00369=377691,340036,804361
BC00370=301973,352945,928572
BC00371=301973,352945,928572
BC00372=301973,352945,928572
BC00373=301973,352945,928572
BC00374=301973,352945,928572
BC00375=301973,352945,928572
BC00376=301974,352945,928571
BC00377=301973,352945,928572
BC00378=301973,352945,928572
BC00379=305078,353410,929381
BC00380=305078,353410,929381
BC00381=305078,353410,929381
BC00382=305078,353410,929381
BC00383=305078,353410,929381
BC00384=305078,353410,929381
BC00385=305078,353410,929381
BC00386=305078,353410,929381
BC00387=355079,392127,745599
BC00388=333047,392127,745599
BC00389=333047,392127,745599
BC00390=333047,392127,745599
BC00391=333047,392127,745599
BC00392=333047,392127,745599
BC00393=333047,392127,745599
BC00394=333047,392127,745599
BC00395=333047,392127,745599
BC00396=333047,392127,745599
BC00397=333047,392127,745599
BC00398=333047,392127,745599
BC00399=333047,392127,745599
BC00400=333047,392127,745599
BC00401=333047,392127,745599
BC00402=330711,385408,779676
BC00403=330711,385408,779676
BC00404=330711,385408,779676
BC00405=330711,385408,779676
BC00406=330711,385408,779676
BC00407=330711,385408,779676
BC00408=330711,385408,779676
BC00409=286508,385408,779676
BC00410=286508,385408,779676
BC00411=286508,385408,779676
BC00412=286508,385408,779676
BC00413=286508,385408,779676
BC00414=286508,385408,779676
BC00415=288154,385206,781872
BC00416=288360,385181,782147
BC00417=288360,385181,782147
BC00418=340469,375654,887477
BC00419=340973,375751,888339
BC00420=340973,375751,888339
BC00421=341056,375767,888482
BC00422=341056,375767,888482
BC00423=341056,375767,888482
BC00424=303693,363347,778304
BC00425=303693,363347,778304
BC00426=303693,363348,778302
BC00427=303693,363347,778303
BC00428=303693,363347,778304
BC00429=303693,363347,778304
BC00430=304263,355192,768709
BC00431=304263,355192,768709
BC00432=304263,355192,768709
BC00433=304263,355192,768709
BC00434=304263,355192,768709
BC00435=304263,355192,768709
BC00436=307126,354525,782310
BC00437=313370,353070,811970
BC00438=313370,353070,811970
BC00439=313370,353070,811970
BC00440=313370,353070,811970
BC00441=313370,353070,811970
BC00442=381578,331383,767352
BC00443=381578,331383,767352
BC00444=381578,331383,767352
BC00445=381578,331383,767352
BC00446=381578,331383,767352
BC00447=381578,331383,767352
BC00448=337601,317122,860141
BC00449=333177,303767,911398
BC00450=333177,303767,911398
BC00451=353932,303767,911398
BC00452=353932,303767,911398
BC00453=333177,303767,911398
BC00454=333177,303767,911398
BC00455=313597,315083,952947
BC00456=313597,315083,952947
BC00457=313597,315083,952947
BC00458=313597,315083,952947
BC00459=313597,315083,952947
BC00460=313597,315083,952947
BC00461=317033,330359,927586
BC00462=204139,405669,1028194
BC00463=121307,427031,1056816
BC00464=21523,502292,1072610
EC00000=-1108551,372643
EC00001=-1108551,372643
EC00002=-1108551,372643
EC00003=-1108551,372643
EC00004=-1108551,372643
EC00005=-1108551,372643
EC00006=-1108551,372643
EC00007=-1108551,372643
EC00008=-1108551,372643
EC00009=-1108551,372643
EC00010=-1108551,372643
EC00011=-1108551,372643
EC00012=-1108551,372643
EC00013=-1108551,372643
EC00014=-1108551,372643
EC00015=-1108551,372643
EC00016=-1108551,372643
EC00017=-1108551,372643
EC00018=-1108551,372643
EC00019=-1108551,372643
EC00020=-1108551,372643
EC00021=-1108551,372643
EC00022=-1108551,372643
EC00023=-1108551,372643
EC00024=-1108551,372643
EC00025=-1108551,372643
EC00026=-1108551,372643
EC00027=-1108551,372643
EC00028=-1108551,372643
EC00029=-1108551,372643
EC00030=-1108551,372643
EC00031=-1108551,372643
EC00032=-1108551,372643
EC00033=-1108551,372643
EC00034=-1108551,372643
EC00035=-1108551,372643
EC00036=-1108551,372643
EC00037=-1108551,372643
EC00038=-1108551,372643
EC00039=-1108551,372643
EC00040=-1108551,372643
EC00041=-1108551,372643
EC00042=-1108551,372643
EC00043=-1108551,372643
EC00044=-1108551,372643
EC00045=-1108551,372643
EC00046=-1108551,372643
EC00047=-1108551,372643
EC00048=-1108551,372643
EC00049=-1108551,372643
EC00050=-1108551,372643
EC00051=-1108551,372643
EC00052=-1108551,372643
EC00053=-1108551,372643
EC00054=-1108551,372643
EC00055=-1108551,372643
EC00056=-1108551,372643
EC00057=-1108551,372643
EC00058=-1108551,372643
EC00059=-1108551,372643
EC00060=-1108551,372643
EC00061=-1108551,372643
EC00062=-1108551,372643
EC00063=-1108551,372643
EC00064=-1108551,372643
EC00065=-1108551,372643
EC00066=-1108551,372643
EC00067=-1108551,372643
EC00068=-1108551,372643
EC00069=-1108551,372643
EC00070=-1108550,372643
EC00071=-1108551,372643
EC00072=-1108551,372643
EC00073=-1108551,372643
EC00074=-1108551,372643
EC00075=-1108551,372643
EC00076=-1108551,372643
EC00077=-1108551,372643
EC00078=-1108551,372643
EC00079=-1108551,372643
EC00080=-1108551,372643
EC00081=-1108551,372643
EC00082=-1108551,372643
EC00083=-1108551,372643
EC00084=-1108551,372643
EC00085=-1108551,372643
EC00086=-1108551,372643
EC00087=-1108551,372643
EC00088=-1108551,372643
EC00089=-1108551,372643
EC00090=-1108551,372643
EC00091=-1108551,372643
EC00092=-1108551,372643
EC00093=-1108551,372643
EC00094=-1108551,372643
EC00095=-1108551,372643
EC00096=-1108551,372643
EC00097=-1108551,372643
EC00098=-1108551,372643
EC00099=-1108551,372643
EC00100=-1108551,372643
EC00101=-1108551,372643
EC00102=-1108551,372643
EC00103=-1108551,372643
EC00104=-1108551,372643
EC00105=-1108551,372643
EC00106=-1108551,372643
EC00107=-1108551,372643
EC00108=-1108551,372643
EC00109=-1108550,372642
EC00110=-1108551,372643
EC00111=-1108551,372643
EC00112=-1108551,372643
EC00113=-1108551,372643
EC00114=-1108551,372643
EC00115=-1108551,372643
EC00116=-1108551,372643
EC00117=-1108551,372643
EC00118=-1108551,372643
EC00119=-1108551,372643
EC00120=-1108551,372643
EC00121=-1108551,372643
EC00122=-1108551,372643
EC00123=-1108551,372643
EC00124=-1108551,372642
EC00125=-1108551,372643
EC00126=-1108551,372643
EC00127=-1108551,372643
EC00128=-1108551,372643
EC00129=-1108551,372643
EC00130=-1108551,372643
EC00131=-1108551,372643
EC00132=-1108551,372643
EC00133=-1108551,372643
EC00134=-1108551,372643
EC00135=-1108551,372643
EC00136=-1108551,372643
EC00137=-1108551,372643
EC00138=-1108551,372643
EC00139=-1108551,372643
EC00140=-1108551,372643
EC00141=-1108551,372643
EC00142=-1108551,372643
EC00143=-1108551,372643
EC00144=-1108551,372643
EC00145=-1108551,372643
EC00146=-1108551,372643
EC00147=-1108551,372643
EC00148=-1108551,372643
EC00149=-1108551,372643
EC00150=-1108551,372643
EC00151=-1108551,372643
EC00152=-1108551,372643
EC00153=-1108551,372643
EC00154=-1108551,372643
EC00155=-1108551,372643
EC00156=-1108551,372643
EC00157=-1108551,372643
EC00158=-1108551,372643
EC00159=-1108551,372643
EC00160=-1108551,372643
EC00161=-1108551,372643
EC00162=-1108551,372643
EC00163=-1108551,372643
EC00164=-1108551,372643
EC00165=-1108551,372643
EC00166=-1108550,372643
EC00167=-1108550,372643
EC00168=-1108551,372643
EC00169=-1108551,372643
EC00170=-1108551,372643
EC00171=-1108551,372643
EC00172=-1108551,372643
EC00173=-1108551,372643
EC00174=-1108551,372643
EC00175=-1108551,372643
EC00176=-1108551,372643
EC00177=-1108551,372643
EC00178=-1108551,372643
EC00179=-1108551,372643
EC00180=-1108551,372643
EC00181=-1108551,372643
EC00182=-1108551,372643
EC00183=-1108551,372643
EC00184=-1108551,372643
EC00185=-1108551,372643
EC00186=-1108550,372643
EC00187=-1108551,372643
EC00188=-1108551,372643
EC00189=-1108551,372643
EC00190=-1108551,372643
EC00191=-1108551,372643
EC00192=-1108551,372643
EC00193=-1108551,372643
EC00194=-1108551,372643
EC00195=-1108551,372643
EC00196=-1108551,372643
EC00197=-1108551,372643
EC00198=-1108551,372643
EC00199=-1108551,372643
EC00200=-1108551,372643
EC00201=-1108551,372643
EC00202=1108549,-740306
EC00203=1108550,-740307
EC00204=1108551,-740307
EC00205=1108551,-740307
EC00206=1108551,-740307
EC00207=1108551,-740307
EC00208=1108551,-740307
EC00209=1108551,-740307
EC00210=1108551,-740307
EC00211=1108551,-740307
EC00212=1108551,-740307
EC00213=1108551,-740307
EC00214=1108551,-740307
EC00215=1108551,-740307
EC00216=1108551,-740307
EC00217=1108551,-740307
EC00218=1108551,-740307
EC00219=1108551,-740307
EC00220=1108551,-740307
EC00221=1108551,-740307
EC00222=1108551,-740307
EC00223=1108551,-740307
EC00224=1108551,-740307
EC00225=1108551,-740307
EC00226=1108551,-740307
EC00227=1108551,-740307
EC00228=1108551,-740307
EC00229=1108551,-740307
EC00230=1108551,-740307
EC00231=1108551,-740307
EC00232=1108551,-740307
EC00233=1108551,-740307
EC00234=1108551,-740307
EC00235=1108551,-740307
EC00236=1108551,-740307
EC00237=1108551,-740307
EC00238=1108551,-740307
EC00239=1108551,-740307
EC00240=1108551,-740307
EC00241=1108551,-740307
EC00242=1108551,-740307
EC00243=1108550,-740307
EC00244=1108551,-740307
EC00245=1108551,-740307
EC00246=1108551,-740307
EC00247=1108551,-740307
EC00248=1108551,-740307
EC00249=1108551,-740307
EC00250=1108551,-740307
EC00251=1108551,-740307
EC00252=1108551,-740307
EC00253=1108551,-740307
EC00254=1108551,-740307
EC00255=1108551,-740307
EC00256=1108551,-740307
EC00257=1108551,-740307
EC00258=1108551,-740307
EC00259=1108551,-740307
EC00260=1108551,-740307
EC00261=1108551,-740307
EC00262=1108551,-740307
EC00263=1108551,-740307
EC00264=1108551,-740307
EC00265=1108551,-740307
EC00266=1108551,-740307
EC00267=1108551,-740307
EC00268=1108551,-740307
EC00269=1108551,-740307
EC00270=1108551,-740307
EC00271=1108551,-740307
EC00272=1108551,-740307
EC00273=1108551,-740307
EC00274=1108551,-740307
EC00275=1108551,-740307
EC00276=1108551,-740307
EC00277=1108551,-740307
EC00278=1108551,-740307
EC00279=1108551,-740307
EC00280=1108551,-740307
EC00281=1108551,-740307
EC00282=1108551,-740307
EC00283=1108551,-740307
EC00284=1108551,-740307
EC00285=1108551,-740307
EC00286=1108549,-740308
EC00287=1108549,-740308
EC00288=1108549,-740308
EC00289=1108549,-740308
EC00290=1108549,-740308
EC00291=1108549,-740308
EC00292=1108550,-740308
EC00293=1108551,-740307
EC00294=1108551,-740307
EC00295=1108548,-740307
EC00296=1108550,-740308
EC00297=1108551,-740307
EC00298=1108551,-740307
EC00299=1108551,-740307
EC00300=1108551,-740307
EC00301=1108551,-740307
EC00302=1108551,-740307
EC00303=1108551,-740307
EC00304=1108551,-740307
EC00305=1108551,-740307
EC00306=1108551,-740307
EC00307=1108551,-740307
EC00308=1108551,-740307
EC00309=1108551,-740307
EC00310=1108551,-740307
EC00311=1108551,-740307
EC00312=1108549,-740308
EC00313=1108550,-740307
EC00314=1108550,-740307
EC00315=1108550,-740307
EC00316=1108551,-740307
EC00317=1108551,-740307
EC00318=1108551,-740307
EC00319=1108551,-740307
EC00320=1108551,-740307
EC00321=1108551,-740307
EC00322=1108551,-740307
EC00323=1108551,-740307
EC00324=1108551,-740307
EC00325=1108551,-740307
EC00326=1108551,-740307
EC00327=1108551,-740307
EC00328=1108551,-740307
EC00329=1108550,-740306
EC00330=1108550,-740306
EC00331=1108549,-740306
EC00332=1108550,-740306
EC00333=1108550,-740306
EC00334=1108550,-740306
EC00335=1108551,-740307
EC00336=1108551,-740307
EC00337=1108551,-740307
EC00338=1108551,-740307
EC00339=1108551,-740307
EC00340=1108551,-740307
EC00341=1108551,-740307
EC00342=1108551,-740307
EC00343=1108551,-740307
EC00344=1108551,-740307
EC00345=1108551,-740307
EC00346=1108551,-740307
EC00347=1108551,-740307
EC00348=1108551,-740307
EC00349=1108551,-740307
EC00350=1108551,-740307
EC00351=1108551,-740307
EC00352=1108551,-740307
EC00353=1108551,-740307
EC00354=1108551,-740307
EC00355=1108551,-740307
EC00356=1108551,-740307
EC00357=1108551,-740307
EC00358=1108551,-740307
EC00359=1108551,-740307
EC00360=1108551,-740307
EC00361=1108551,-740307
EC00362=1108551,-740307
EC00363=1108551,-740307
EC00364=1108551,-740307
EC00365=1108551,-740307
EC00366=1108551,-740307
EC00367=1108551,-740307
EC00368=1108551,-740307
EC00369=1108551,-740307
EC00370=1108551,-740307
EC00371=1108551,-740307
EC00372=1108551,-740307
EC00373=1108551,-740307
EC00374=1108551,-740307
EC00375=1108551,-740307
EC00376=1108550,-740307
EC00377=1108551,-740307
EC00378=1108551,-740307
EC00379=1108551,-740307
EC00380=1108551,-740307
EC00381=1108551,-740307
EC00382=1108551,-740307
EC00383=1108551,-740307
EC00384=1108551,-740307
EC00385=1108551,-740307
EC00386=1108551,-740307
EC00387=1108551,-740307
EC00388=1108551,-740307
EC00389=1108551,-740307
EC00390=1108551,-740307
EC00391=1108551,-740307
EC00392=1108551,-740307
EC00393=1108551,-740307
EC00394=1108551,-740307
EC00395=1108551,-740307
EC00396=1108551,-740307
EC00397=1108551,-740307
EC00398=1108551,-740307
EC00399=1108551,-740307
EC00400=1108551,-740307
EC00401=1108551,-740307
EC00402=1108551,-740307
EC00403=1108551,-740307
EC00404=1108551,-740307
EC00405=1108551,-740307
EC00406=1108551,-740307
EC00407=1108551,-740307
EC00408=1108551,-740307
EC00409=1108551,-740307
EC00410=1108551,-740307
EC00411=1108551,-740307
EC00412=1108551,-740307
EC00413=1108551,-740307
EC00414=1108551,-740307
EC00415=1108551,-740307
EC00416=1108551,-740307
EC00417=1108551,-740307
EC00418=1108549,-740308
EC00419=1108549,-740308
EC00420=1108549,-740308
EC00421=1108549,-740308
EC00422=1108549,-740308
EC00423=1108549,-740308
EC00424=1108551,-740307
EC00425=1108551,-740307
EC00426=1108548,-740307
EC00427=1108550,-740308
EC00428=1108551,-740307
EC00429=1108551,-740307
EC00430=1108551,-740307
EC00431=1108551,-740307
EC00432=1108551,-740307
EC00433=1108551,-740307
EC00434=1108551,-740307
EC00435=1108551,-740307
EC00436=1108551,-740307
EC00437=1108551,-740307
EC00438=1108551,-740307
EC00439=1108551,-740307
EC00440=1108551,-740307
EC00441=1108551,-740307
EC00442=1108551,-740307
EC00443=1108551,-740307
EC00444=1108551,-740307
EC00445=1108551,-740307
EC00446=1108551,-740307
EC00447=1108551,-740307
EC00448=1108551,-740307
EC00449=1108551,-740307
EC00450=1108551,-740307
EC00451=1108551,-740307
EC00452=1108551,-740307
EC00453=1108551,-740307
EC00454=1108551,-740307
EC00455=1108551,-740307
EC00456=1108551,-740307
EC00457=1108551,-740307
EC00458=1108551,-740307
EC00459=1108551,-740307
EC00460=1108551,-740307
EC00461=1108551,-740307
EC00462=1108551,-740307
EC00463=1108551,-740307
EC00464=1108551,-740307
///POSTYPE BASE
///RECTAN
///RCONF 0,0,0,0,1,0,0,0,0,0,0,0,0,0,0,0,0,0,0,0,0,0,0,0
P00006=2.006,1.622,-0.565,0.0000,0.0000,0.0000
P00021=0.073,2.058,-0.109,0.0000,0.0000,0.0000
P00022=2.006,1.622,-0.565,0.0000,0.0000,0.0000
///RCONF 0,0,0,0,0,0,0,0,0,0,0,0,0,0,0,0,0,0,0,0,0,0,0,0
P00023=-2.957,-4.083,2.762,0.0000,0.0000,0.0000
P00024=-1.466,-0.226,-0.419,0.0000,0.0000,0.0000
P00025=3.643,0.007,-2.585,0.0000,0.0000,0.0000
P00026=2.644,0.055,-2.583,0.0000,0.0000,0.0000
P00027=2.278,0.099,-4.210,0.0000,0.0000,0.0000
P00028=-1.778,-0.182,-2.050,0.0000,0.0000,0.0000
P00029=1.749,4.006,-0.261,0.0000,0.0000,0.0000
P00030=-0.014,-0.768,0.131,0.0000,0.0000,0.0000
P00031=-0.170,0.039,-0.647,0.0000,0.0000,0.0000
P00032=-0.423,0.157,3.222,0.0000,0.0000,0.0000
P00033=0.854,-1.099,3.047,0.0000,0.0000,0.0000
P00041=-0.109,0.014,0.966,0.0000,0.0000,0.0000
P00042=-0.220,0.371,-0.613,0.0000,0.0000,0.0000
P00045=-8.836,-6.632,-1.438,0.0000,0.0000,0.0000
P00046=-7.725,-0.107,-2.878,0.0000,0.0000,0.0000
///RCONF 0,1,0,0,0,0,0,0,0,0,0,0,0,0,0,0,0,0,0,0,0,0,0,0
P00047=0.052,4.745,-6.175,0.0000,0.0000,0.0000
///RCONF 0,0,0,0,0,0,0,0,0,0,0,0,0,0,0,0,0,0,0,0,0,0,0,0
P00048=-10.315,0.035,-3.101,0.0000,0.0000,0.0000
P00050=-0.123,2.174,-1.314,0.0000,0.0000,0.0000
P00051=-5.945,4.696,-10.293,0.0000,0.0000,0.0000
P00052=-0.153,5.586,-7.982,0.0000,0.0000,0.0000
P00053=0.015,-0.644,-4.942,0.0000,0.0000,0.0000
//INST
///DATE 2024/12/18 19:45
///ATTR SC,RW
///GROUP1 RB1,BS1
///GROUP2 ST1
NOP
'X2_100(P)(125,-90)
COMM PAUSE
COMM MOVJ C00000 BC00000 VJ=20.00  +MOVJ EC00000 VJ=20.00
COMM MOVJ C00001 BC00001 VJ=20.00  +MOVJ EC00001 VJ=20.00
COMM PAUSE
COMM PAUSE
COMM '
COMM MOVJ C00002 BC00002 VJ=100.00  +MOVJ EC00002 VJ=100.00
COMM MOVJ C00003 BC00003 VJ=100.00  +MOVJ EC00003 VJ=100.00
COMM '
COMM MOVJ C00004 BC00004 VJ=100.00  +MOVJ EC00004 VJ=100.00
COMM MOVJ C00005 BC00005 VJ=100.00  +MOVJ EC00005 VJ=100.00
COMM MOVJ C00006 BC00006 VJ=100.00  +MOVJ EC00006 VJ=100.00
COMM MOVJ C00007 BC00007 VJ=100.00  +MOVJ EC00007 VJ=100.00
COMM MOVJ C00008 BC00008 VJ=100.00  +MOVJ EC00008 VJ=100.00
COMM 'Path S3336
COMM SFTOF3D
COMM MOVJ C00009 BC00009 VJ=100.00  +MOVJ EC00009 VJ=100.00
COMM MOVL C00010 BC00010 V=800.0  +MOVJ EC00010 VJ=100.00
COMM SMOVL C00011 BC00011 V=166.7  +MOVJ EC00011
COMM SREFP 3 C00012 BC00012  +REFP EC00012
COMM CALL JOB:SEARCH-R1-S13D
COMM SET P021 P006
COMM SFTON3D P021
COMM SMOVL C00013 BC00013 V=166.7  +MOVJ EC00013
COMM SREFP 3 C00014 BC00014  +REFP EC00014
COMM CALL JOB:SEARCH-R1-S13D
COMM SET P021 P006
COMM SFTON3D P021
COMM SMOVL C00015 BC00015 V=166.7  +MOVJ EC00015
COMM MOVL C00016 BC00016 V=1000.0  +MOVJ EC00016 VJ=100.00
COMM 'EndPath S3336
COMM 'Path S3337
COMM SFTOF3D
COMM MOVJ C00017 BC00017 VJ=100.00  +MOVJ EC00017 VJ=100.00
COMM MOVL C00018 BC00018 V=800.0  +MOVJ EC00018 VJ=100.00
COMM SMOVL C00019 BC00019 V=166.7  +MOVJ EC00019
COMM SREFP 3 C00020 BC00020  +REFP EC00020
COMM CALL JOB:SEARCH-R1-S13D
COMM SET P022 P006
COMM SFTON3D P022
COMM SMOVL C00021 BC00021 V=166.7  +MOVJ EC00021
COMM SREFP 3 C00022 BC00022  +REFP EC00022
COMM CALL JOB:SEARCH-R1-S13D
COMM SET P022 P006
COMM SFTON3D P022
COMM SMOVL C00023 BC00023 V=166.7  +MOVJ EC00023
COMM MOVL C00024 BC00024 V=1000.0  +MOVJ EC00024 VJ=100.00
COMM 'EndPath S3337
COMM 'Path S3338
COMM SFTOF3D
COMM MOVJ C00025 BC00025 VJ=100.00  +MOVJ EC00025 VJ=100.00
COMM MOVL C00026 BC00026 V=800.0  +MOVJ EC00026 VJ=100.00
COMM SMOVL C00027 BC00027 V=166.7  +MOVJ EC00027
COMM SREFP 3 C00028 BC00028  +REFP EC00028
COMM CALL JOB:SEARCH-R1-S13D
COMM SET P023 P006
COMM SFTON3D P023
COMM SMOVL C00029 BC00029 V=166.7  +MOVJ EC00029
COMM SREFP 3 C00030 BC00030  +REFP EC00030
COMM CALL JOB:SEARCH-R1-S13D
COMM SET P023 P006
COMM SFTON3D P023
COMM SMOVL C00031 BC00031 V=166.7  +MOVJ EC00031
COMM MOVL C00032 BC00032 V=1000.0  +MOVJ EC00032 VJ=100.00
COMM 'EndPath S3338
COMM MOVJ C00033 BC00033 VJ=100.00  +MOVJ EC00033 VJ=100.00
COMM 'Path S3339
COMM SFTOF3D
COMM MOVJ C00034 BC00034 VJ=100.00  +MOVJ EC00034 VJ=100.00
COMM MOVL C00035 BC00035 V=800.0  +MOVJ EC00035 VJ=100.00
COMM SMOVL C00036 BC00036 V=166.7  +MOVJ EC00036
COMM SREFP 3 C00037 BC00037  +REFP EC00037
COMM CALL JOB:SEARCH-R1-S13D
COMM SET P024 P006
COMM SFTON3D P024
COMM SMOVL C00038 BC00038 V=166.7  +MOVJ EC00038
COMM SREFP 3 C00039 BC00039  +REFP EC00039
COMM CALL JOB:SEARCH-R1-S13D
COMM SET P024 P006
COMM SFTON3D P024
COMM SMOVL C00040 BC00040 V=166.7  +MOVJ EC00040
COMM MOVL C00041 BC00041 V=1000.0  +MOVJ EC00041 VJ=100.00
COMM 'EndPath S3339
COMM 'Path S3341
COMM SFTOF3D
COMM MOVJ C00042 BC00042 VJ=100.00  +MOVJ EC00042 VJ=100.00
COMM MOVL C00043 BC00043 V=800.0  +MOVJ EC00043 VJ=100.00
COMM SMOVL C00044 BC00044 V=166.7  +MOVJ EC00044
COMM SREFP 3 C00045 BC00045  +REFP EC00045
COMM CALL JOB:SEARCH-R1-S13D
COMM SET P025 P006
COMM SFTON3D P025
COMM SMOVL C00046 BC00046 V=166.7  +MOVJ EC00046
COMM SREFP 3 C00047 BC00047  +REFP EC00047
COMM CALL JOB:SEARCH-R1-S13D
COMM SET P025 P006
COMM SFTON3D P025
COMM SMOVL C00048 BC00048 V=166.7  +MOVJ EC00048
COMM MOVL C00049 BC00049 V=1000.0  +MOVJ EC00049 VJ=100.00
COMM 'EndPath S3341
COMM 'Path S3343
COMM SFTOF3D
COMM MOVJ C00050 BC00050 VJ=100.00  +MOVJ EC00050 VJ=100.00
COMM MOVL C00051 BC00051 V=800.0  +MOVJ EC00051 VJ=100.00
COMM SMOVL C00052 BC00052 V=166.7  +MOVJ EC00052
COMM SREFP 3 C00053 BC00053  +REFP EC00053
COMM CALL JOB:SEARCH-R1-S13D
COMM SET P026 P006
COMM SFTON3D P026
COMM SMOVL C00054 BC00054 V=166.7  +MOVJ EC00054
COMM SREFP 3 C00055 BC00055  +REFP EC00055
COMM CALL JOB:SEARCH-R1-S13D
COMM SET P026 P006
COMM SFTON3D P026
COMM SMOVL C00056 BC00056 V=166.7  +MOVJ EC00056
COMM MOVL C00057 BC00057 V=1000.0  +MOVJ EC00057 VJ=100.00
COMM 'EndPath S3343
COMM MOVJ C00058 BC00058 VJ=100.00  +MOVJ EC00058 VJ=100.00
COMM 'Path S3345
COMM SFTOF3D
COMM MOVJ C00059 BC00059 VJ=100.00  +MOVJ EC00059 VJ=100.00
COMM MOVL C00060 BC00060 V=800.0  +MOVJ EC00060 VJ=100.00
COMM SMOVL C00061 BC00061 V=166.7  +MOVJ EC00061
COMM SREFP 3 C00062 BC00062  +REFP EC00062
COMM CALL JOB:SEARCH-R1-S13D
COMM SET P027 P006
COMM SFTON3D P027
COMM SMOVL C00063 BC00063 V=166.7  +MOVJ EC00063
COMM SREFP 3 C00064 BC00064  +REFP EC00064
COMM CALL JOB:SEARCH-R1-S13D
COMM SET P027 P006
COMM SFTON3D P027
COMM SMOVL C00065 BC00065 V=166.7  +MOVJ EC00065
COMM MOVL C00066 BC00066 V=1000.0  +MOVJ EC00066 VJ=100.00
COMM 'EndPath S3345
COMM MOVJ C00067 BC00067 VJ=100.00  +MOVJ EC00067 VJ=100.00
COMM 'Path S3347
COMM SFTOF3D
COMM MOVJ C00068 BC00068 VJ=100.00  +MOVJ EC00068 VJ=100.00
COMM MOVL C00069 BC00069 V=800.0  +MOVJ EC00069 VJ=100.00
COMM SMOVL C00070 BC00070 V=166.7  +MOVJ EC00070
COMM SREFP 3 C00071 BC00071  +REFP EC00071
COMM CALL JOB:SEARCH-R1-S13D
COMM SET P028 P006
COMM SFTON3D P028
COMM SMOVL C00072 BC00072 V=166.7  +MOVJ EC00072
COMM SREFP 3 C00073 BC00073  +REFP EC00073
COMM CALL JOB:SEARCH-R1-S13D
COMM SET P028 P006
COMM SFTON3D P028
COMM SMOVL C00074 BC00074 V=166.7  +MOVJ EC00074
COMM MOVL C00075 BC00075 V=1000.0  +MOVJ EC00075 VJ=100.00
COMM 'EndPath S3347
COMM 'Path S3349
COMM SFTOF3D
COMM MOVJ C00076 BC00076 VJ=100.00  +MOVJ EC00076 VJ=100.00
COMM MOVL C00077 BC00077 V=800.0  +MOVJ EC00077 VJ=100.00
COMM SMOVL C00078 BC00078 V=166.7  +MOVJ EC00078
COMM SREFP 3 C00079 BC00079  +REFP EC00079
COMM CALL JOB:SEARCH-R1-S13D
COMM SET P029 P006
COMM SFTON3D P029
COMM SMOVL C00080 BC00080 V=166.7  +MOVJ EC00080
COMM SREFP 3 C00081 BC00081  +REFP EC00081
COMM CALL JOB:SEARCH-R1-S13D
COMM SET P029 P006
COMM SFTON3D P029
COMM SMOVL C00082 BC00082 V=166.7  +MOVJ EC00082
COMM MOVL C00083 BC00083 V=1000.0  +MOVJ EC00083 VJ=100.00
COMM 'EndPath S3349
COMM 'Path S3350
COMM SFTOF3D
COMM MOVJ C00084 BC00084 VJ=100.00  +MOVJ EC00084 VJ=100.00
COMM MOVL C00085 BC00085 V=800.0  +MOVJ EC00085 VJ=100.00
COMM SMOVL C00086 BC00086 V=166.7  +MOVJ EC00086
COMM SREFP 3 C00087 BC00087  +REFP EC00087
COMM CALL JOB:SEARCH-R1-S13D
COMM SET P030 P006
COMM SFTON3D P030
COMM SMOVL C00088 BC00088 V=166.7  +MOVJ EC00088
COMM SREFP 3 C00089 BC00089  +REFP EC00089
COMM CALL JOB:SEARCH-R1-S13D
COMM SET P030 P006
COMM SFTON3D P030
COMM SMOVL C00090 BC00090 V=166.7  +MOVJ EC00090
COMM SMOVL C00091 BC00091 V=166.7  +MOVJ EC00091
COMM SREFP 3 C00092 BC00092  +REFP EC00092
COMM CALL JOB:SEARCH-R1-S13D
COMM SET P030 P006
COMM SFTON3D P030
COMM SMOVL C00093 BC00093 V=166.7  +MOVJ EC00093
COMM MOVL C00094 BC00094 V=1000.0  +MOVJ EC00094 VJ=100.00
COMM 'EndPath S3350
COMM 'Path S3351
COMM SFTOF3D
COMM MOVJ C00095 BC00095 VJ=100.00  +MOVJ EC00095 VJ=100.00
COMM MOVL C00096 BC00096 V=800.0  +MOVJ EC00096 VJ=100.00
COMM SMOVL C00097 BC00097 V=166.7  +MOVJ EC00097
COMM SREFP 3 C00098 BC00098  +REFP EC00098
COMM CALL JOB:SEARCH-R1-S13D
COMM SET P031 P006
COMM SFTON3D P031
COMM SMOVL C00099 BC00099 V=166.7  +MOVJ EC00099
COMM SREFP 3 C00100 BC00100  +REFP EC00100
COMM CALL JOB:SEARCH-R1-S13D
COMM SET P031 P006
COMM SFTON3D P031
COMM SMOVL C00101 BC00101 V=166.7  +MOVJ EC00101
COMM MOVL C00102 BC00102 V=1000.0  +MOVJ EC00102 VJ=100.00
COMM 'EndPath S3351
COMM MOVJ C00103 BC00103 VJ=100.00  +MOVJ EC00103 VJ=100.00
COMM 'Path S3352
COMM SFTOF3D
COMM MOVJ C00104 BC00104 VJ=100.00  +MOVJ EC00104 VJ=100.00
COMM MOVL C00105 BC00105 V=800.0  +MOVJ EC00105 VJ=100.00
COMM SMOVL C00106 BC00106 V=166.7  +MOVJ EC00106
COMM SREFP 3 C00107 BC00107  +REFP EC00107
COMM CALL JOB:SEARCH-R1-S13D
COMM SET P032 P006
COMM SFTON3D P032
COMM SMOVL C00108 BC00108 V=166.7  +MOVJ EC00108
COMM SREFP 3 C00109 BC00109  +REFP EC00109
COMM CALL JOB:SEARCH-R1-S13D
COMM SET P032 P006
COMM SFTON3D P032
COMM SMOVL C00110 BC00110 V=166.7  +MOVJ EC00110
COMM MOVL C00111 BC00111 V=1000.0  +MOVJ EC00111 VJ=100.00
COMM 'EndPath S3352
COMM 'Path S3353
COMM SFTOF3D
COMM MOVJ C00112 BC00112 VJ=100.00  +MOVJ EC00112 VJ=100.00
COMM MOVL C00113 BC00113 V=800.0  +MOVJ EC00113 VJ=100.00
COMM SMOVL C00114 BC00114 V=166.7  +MOVJ EC00114
COMM SREFP 3 C00115 BC00115  +REFP EC00115
COMM CALL JOB:SEARCH-R1-S13D
COMM SET P033 P006
COMM SFTON3D P033
COMM SMOVL C00116 BC00116 V=166.7  +MOVJ EC00116
COMM SREFP 3 C00117 BC00117  +REFP EC00117
COMM CALL JOB:SEARCH-R1-S13D
COMM SET P033 P006
COMM SFTON3D P033
COMM SMOVL C00118 BC00118 V=166.7  +MOVJ EC00118
COMM MOVL C00119 BC00119 V=1000.0  +MOVJ EC00119 VJ=100.00
COMM 'EndPath S3353
COMM MOVJ C00120 BC00120 VJ=100.00  +MOVJ EC00120 VJ=100.00
COMM MOVJ C00121 BC00121 VJ=100.00  +MOVJ EC00121 VJ=100.00
COMM 'Path W3292
COMM SFTOF3D
COMM SFTON3D P021
COMM MOVJ C00122 BC00122 VJ=100.00  +MOVJ EC00122 VJ=100.00
COMM SMOVL C00123 BC00123 V=800.0  +MOVJ EC00123
COMM SMOVL C00124 BC00124 V=166.7 PL=0  +MOVJ EC00124
COMM MACRO1 MJ#(0) ARGF9
COMM ARCON
COMM SMOVL C00125 BC00125 V=11.7  +MOVJ EC00125
COMM SMOVL C00126 BC00126 V=11.7  +MOVJ EC00126
COMM SMOVL C00127 BC00127 V=11.7  +MOVJ EC00127
COMM ARCOF
COMM SMOVL C00128 BC00128 V=800.0  +MOVJ EC00128
COMM SMOVL C00129 BC00129 V=1000.0  +MOVJ EC00129
COMM SFTOF3D
COMM 'EndPath W3292
COMM 'Path W3293
COMM SFTOF3D
COMM SFTON3D P022
COMM MOVJ C00130 BC00130 VJ=100.00  +MOVJ EC00130 VJ=100.00
COMM SMOVL C00131 BC00131 V=800.0  +MOVJ EC00131
COMM SMOVL C00132 BC00132 V=166.7 PL=0  +MOVJ EC00132
COMM ARCON
COMM SMOVL C00133 BC00133 V=11.7  +MOVJ EC00133
COMM ARCOF
COMM SMOVL C00134 BC00134 V=800.0  +MOVJ EC00134
COMM SMOVL C00135 BC00135 V=1000.0  +MOVJ EC00135
COMM SFTOF3D
COMM 'EndPath W3293
COMM 'Path W3294
COMM SFTOF3D
COMM SFTON3D P023
COMM MOVJ C00136 BC00136 VJ=100.00  +MOVJ EC00136 VJ=100.00
COMM SMOVL C00137 BC00137 V=800.0  +MOVJ EC00137
COMM SMOVL C00138 BC00138 V=166.7 PL=0  +MOVJ EC00138
COMM ARCON
COMM SMOVL C00139 BC00139 V=11.7  +MOVJ EC00139
COMM ARCOF
COMM SMOVL C00140 BC00140 V=800.0  +MOVJ EC00140
COMM SMOVL C00141 BC00141 V=1000.0  +MOVJ EC00141
COMM SFTOF3D
COMM 'EndPath W3294
COMM '
COMM MOVJ C00142 BC00142 VJ=100.00  +MOVJ EC00142 VJ=100.00
COMM 'Path W3340
COMM SFTOF3D
COMM SFTON3D P024
COMM MOVJ C00143 BC00143 VJ=100.00  +MOVJ EC00143 VJ=100.00
COMM SMOVL C00144 BC00144 V=800.0  +MOVJ EC00144
COMM SMOVL C00145 BC00145 V=150.0 PL=0  +MOVJ EC00145
COMM ARCON
COMM SMOVL C00146 BC00146 V=11.7  +MOVJ EC00146
COMM SMOVL C00147 BC00147 V=11.7  +MOVJ EC00147
COMM SMOVL C00148 BC00148 V=11.7  +MOVJ EC00148
COMM ARCOF
COMM SMOVL C00149 BC00149 V=800.0  +MOVJ EC00149
COMM SMOVL C00150 BC00150 V=1000.0  +MOVJ EC00150
COMM SFTOF3D
COMM 'EndPath W3340
COMM 'Path W3342
COMM SFTOF3D
COMM SFTON3D P025
COMM MOVJ C00151 BC00151 VJ=100.00  +MOVJ EC00151 VJ=100.00
COMM SMOVL C00152 BC00152 V=800.0  +MOVJ EC00152
COMM SMOVL C00153 BC00153 V=150.0 PL=0  +MOVJ EC00153
COMM ARCON
COMM SMOVL C00154 BC00154 V=11.7  +MOVJ EC00154
COMM ARCOF
COMM SMOVL C00155 BC00155 V=800.0  +MOVJ EC00155
COMM SMOVL C00156 BC00156 V=1000.0  +MOVJ EC00156
COMM SFTOF3D
COMM 'EndPath W3342
COMM 'Path W3344
COMM SFTOF3D
COMM SFTON3D P026
COMM MOVJ C00157 BC00157 VJ=100.00  +MOVJ EC00157 VJ=100.00
COMM SMOVL C00158 BC00158 V=800.0  +MOVJ EC00158
COMM SMOVL C00159 BC00159 V=150.0 PL=0  +MOVJ EC00159
COMM ARCON
COMM SMOVL C00160 BC00160 V=11.7  +MOVJ EC00160
COMM ARCOF
COMM SMOVL C00161 BC00161 V=800.0  +MOVJ EC00161
COMM SMOVL C00162 BC00162 V=1000.0  +MOVJ EC00162
COMM SFTOF3D
COMM 'EndPath W3344
COMM '
COMM MOVJ C00163 BC00163 VJ=100.00  +MOVJ EC00163 VJ=100.00
COMM 'Path W3346
COMM SFTOF3D
COMM SFTON3D P027
COMM MOVJ C00164 BC00164 VJ=100.00  +MOVJ EC00164 VJ=100.00
COMM SMOVL C00165 BC00165 V=800.0  +MOVJ EC00165
COMM SMOVL C00166 BC00166 V=150.0 PL=0  +MOVJ EC00166
COMM ARCON
COMM SMOVL C00167 BC00167 V=11.7  +MOVJ EC00167
COMM ARCOF
COMM SMOVL C00168 BC00168 V=800.0  +MOVJ EC00168
COMM SMOVL C00169 BC00169 V=1000.0  +MOVJ EC00169
COMM SFTOF3D
COMM 'EndPath W3346
COMM 'Path W3348
COMM SFTOF3D
COMM SFTON3D P028
COMM MOVJ C00170 BC00170 VJ=100.00  +MOVJ EC00170 VJ=100.00
COMM SMOVL C00171 BC00171 V=800.0  +MOVJ EC00171
COMM SMOVL C00172 BC00172 V=150.0 PL=0  +MOVJ EC00172
COMM ARCON
COMM SMOVL C00173 BC00173 V=11.7  +MOVJ EC00173
COMM ARCOF
COMM SMOVL C00174 BC00174 V=800.0  +MOVJ EC00174
COMM SMOVL C00175 BC00175 V=1000.0  +MOVJ EC00175
COMM SFTOF3D
COMM 'EndPath W3348
COMM 'Path W3350
COMM SFTOF3D
COMM SFTON3D P029
COMM MOVJ C00176 BC00176 VJ=100.00  +MOVJ EC00176 VJ=100.00
COMM SMOVL C00177 BC00177 V=800.0  +MOVJ EC00177
COMM SMOVL C00178 BC00178 V=150.0 PL=0  +MOVJ EC00178
COMM ARCON
COMM SMOVL C00179 BC00179 V=11.7  +MOVJ EC00179
COMM SMOVL C00180 BC00180 V=11.7  +MOVJ EC00180
COMM ARCOF
COMM SMOVL C00181 BC00181 V=800.0  +MOVJ EC00181
COMM SMOVL C00182 BC00182 V=1000.0  +MOVJ EC00182
COMM SFTOF3D
COMM 'EndPath W3350
COMM MOVJ C00183 BC00183 VJ=100.00  +MOVJ EC00183 VJ=100.00
COMM '
COMM 'Path W3316
COMM SFTOF3D
COMM SFTON3D P031
COMM MOVJ C00184 BC00184 VJ=100.00  +MOVJ EC00184 VJ=100.00
COMM SMOVL C00185 BC00185 V=800.0  +MOVJ EC00185
COMM SMOVL C00186 BC00186 V=150.0 PL=0  +MOVJ EC00186
COMM MACRO1 MJ#(0) ARGF21
COMM ARCON
COMM SMOVL C00187 BC00187 V=10.0  +MOVJ EC00187
COMM SFTON3D P030
COMM SMOVL C00188 BC00188 V=10.0  +MOVJ EC00188
COMM SMOVL C00189 BC00189 V=10.0  +MOVJ EC00189
COMM ARCOF
COMM SMOVL C00190 BC00190 V=800.0  +MOVJ EC00190
COMM SMOVL C00191 BC00191 V=1000.0  +MOVJ EC00191
COMM SFTOF3D
COMM 'EndPath W3316
COMM MOVJ C00192 BC00192 VJ=100.00  +MOVJ EC00192 VJ=100.00
COMM '
COMM 'Path W3319
COMM SFTOF3D
COMM SFTON3D P032
COMM MOVJ C00193 BC00193 VJ=100.00  +MOVJ EC00193 VJ=100.00
COMM SMOVL C00194 BC00194 V=800.0  +MOVJ EC00194
COMM SMOVL C00195 BC00195 V=150.0 PL=0  +MOVJ EC00195
COMM ARCON
COMM SFTON3D P033
COMM SMOVL C00196 BC00196 V=9.2  +MOVJ EC00196
COMM ARCOF
COMM SMOVL C00197 BC00197 V=800.0  +MOVJ EC00197
COMM SMOVL C00198 BC00198 V=1000.0  +MOVJ EC00198
COMM SFTOF3D
COMM 'EndPath W3319
COMM MOVJ C00199 BC00199 VJ=100.00  +MOVJ EC00199 VJ=100.00
COMM MOVJ C00200 BC00200 VJ=100.00  +MOVJ EC00200 VJ=100.00
COMM '
COMM MOVJ C00201 BC00201 VJ=100.00  +MOVJ EC00201 VJ=100.00
CALL JOB:CLEAN-R1_KM_NEW
MOVJ C00202 BC00202 VJ=15.00  +MOVJ EC00202 VJ=100.00
MOVJ C00203 BC00203 VJ=20.00  +MOVJ EC00203 VJ=20.00
'
'Path S3355
SFTOF3D
MOVJ C00204 BC00204 VJ=15.00  +MOVJ EC00204 VJ=100.00
MOVL C00205 BC00205 V=800.0  +MOVJ EC00205 VJ=100.00
MOVL C00206 BC00206 V=800.0  +MOVJ EC00206 VJ=100.00
SMOVL C00207 BC00207 V=166.7  +MOVJ EC00207
SREFP 3 C00208 BC00208  +REFP EC00208
CALL JOB:SEARCH-R1-S13D
SET P041 P006
SFTON3D P041
SMOVL C00209 BC00209 V=166.7  +MOVJ EC00209
SREFP 3 C00210 BC00210  +REFP EC00210
CALL JOB:SEARCH-R1-S13D
SET P041 P006
SFTON3D P041
SMOVL C00211 BC00211 V=166.7  +MOVJ EC00211
MOVL C00212 BC00212 V=250.0  +MOVJ EC00212 VJ=100.00
'EndPath S3355
'Path S3356
SFTOF3D
MOVJ C00213 BC00213 VJ=100.00  +MOVJ EC00213 VJ=100.00
MOVL C00214 BC00214 V=800.0  +MOVJ EC00214 VJ=100.00
SMOVL C00215 BC00215 V=166.7  +MOVJ EC00215
SREFP 3 C00216 BC00216  +REFP EC00216
CALL JOB:SEARCH-R1-S13D
SET P042 P006
SFTON3D P042
SMOVL C00217 BC00217 V=166.7  +MOVJ EC00217
SREFP 3 C00218 BC00218  +REFP EC00218
CALL JOB:SEARCH-R1-S13D
SET P042 P006
SFTON3D P042
SMOVL C00219 BC00219 V=166.7  +MOVJ EC00219
MOVL C00220 BC00220 V=1000.0  +MOVJ EC00220 VJ=100.00
'EndPath S3356
'EndPath S3357
'Path S3358
SFTOF3D
'EndPath S3358
'Path S3359
SFTOF3D
MOVJ C00221 BC00221 VJ=100.00  +MOVJ EC00221 VJ=100.00
MOVL C00222 BC00222 V=800.0  +MOVJ EC00222 VJ=100.00
SMOVL C00223 BC00223 V=166.7  +MOVJ EC00223
SREFP 3 C00224 BC00224  +REFP EC00224
CALL JOB:SEARCH-R1-S13D
SET P045 P006
SFTON3D P045
SMOVL C00225 BC00225 V=166.7  +MOVJ EC00225
SREFP 3 C00226 BC00226  +REFP EC00226
CALL JOB:SEARCH-R1-S13D
SET P045 P006
SFTON3D P045
SMOVL C00227 BC00227 V=166.7  +MOVJ EC00227
MOVL C00228 BC00228 V=1000.0  +MOVJ EC00228 VJ=100.00
'EndPath S3359
'Path S3360
SFTOF3D
MOVJ C00229 BC00229 VJ=100.00  +MOVJ EC00229 VJ=100.00
MOVL C00230 BC00230 V=800.0  +MOVJ EC00230 VJ=100.00
SMOVL C00231 BC00231 V=166.7  +MOVJ EC00231
SREFP 3 C00232 BC00232  +REFP EC00232
CALL JOB:SEARCH-R1-S13D
SET P046 P006
SFTON3D P046
SMOVL C00233 BC00233 V=166.7  +MOVJ EC00233
SREFP 3 C00234 BC00234  +REFP EC00234
CALL JOB:SEARCH-R1-S13D
SET P046 P006
SFTON3D P046
SMOVL C00235 BC00235 V=166.7  +MOVJ EC00235
MOVL C00236 BC00236 V=1000.0  +MOVJ EC00236 VJ=100.00
'EndPath S3360
MOVJ C00237 BC00237 VJ=100.00  +MOVJ EC00237 VJ=100.00
'Path S3361
SFTOF3D
MOVJ C00238 BC00238 VJ=25.00  +MOVJ EC00238 VJ=100.00
MOVL C00239 BC00239 V=800.0  +MOVJ EC00239 VJ=100.00
SMOVL C00240 BC00240 V=166.7  +MOVJ EC00240
SREFP 3 C00241 BC00241  +REFP EC00241
CALL JOB:SEARCH-R1-S13D
SET P047 P006
SFTON3D P047
SMOVL C00242 BC00242 V=166.7  +MOVJ EC00242
SREFP 3 C00243 BC00243  +REFP EC00243
CALL JOB:SEARCH-R1-S13D
SET P047 P006
SFTON3D P047
SMOVL C00244 BC00244 V=166.7  +MOVJ EC00244
MOVL C00245 BC00245 V=1000.0  +MOVJ EC00245 VJ=100.00
'EndPath S3361
'Path S3362
SFTOF3D
MOVJ C00246 BC00246 VJ=100.00  +MOVJ EC00246 VJ=100.00
MOVL C00247 BC00247 V=800.0  +MOVJ EC00247 VJ=100.00
SMOVL C00248 BC00248 V=166.7  +MOVJ EC00248
SREFP 3 C00249 BC00249  +REFP EC00249
CALL JOB:SEARCH-R1-S13D
SET P048 P006
SFTON3D P048
SMOVL C00250 BC00250 V=166.7  +MOVJ EC00250
SREFP 3 C00251 BC00251  +REFP EC00251
CALL JOB:SEARCH-R1-S13D
SET P048 P006
SFTON3D P048
SMOVL C00252 BC00252 V=166.7  +MOVJ EC00252
MOVL C00253 BC00253 V=1000.0  +MOVJ EC00253 VJ=100.00
MOVJ C00254 BC00254 VJ=15.00  +MOVJ EC00254 VJ=15.00
'EndPath S3362
'Path S3363
SFTOF3D
MOVJ C00255 BC00255 VJ=20.00  +MOVJ EC00255 VJ=100.00
MOVJ C00256 BC00256 VJ=25.00  +MOVJ EC00256 VJ=100.00
MOVL C00257 BC00257 V=800.0  +MOVJ EC00257 VJ=100.00
SMOVL C00258 BC00258 V=166.7  +MOVJ EC00258
SREFP 3 C00259 BC00259  +REFP EC00259
CALL JOB:SEARCH-R1-S13D
SET P050 P006
SFTON3D P050
SMOVL C00260 BC00260 V=166.7  +MOVJ EC00260
SREFP 3 C00261 BC00261  +REFP EC00261
CALL JOB:SEARCH-R1-S13D
SET P050 P006
SFTON3D P050
SMOVL C00262 BC00262 V=166.7  +MOVJ EC00262
'EndPath S3364
'Path S3365
SFTOF3D
MOVL C00263 BC00263 V=800.0  +MOVJ EC00263 VJ=100.00
SMOVL C00264 BC00264 V=166.7  +MOVJ EC00264
SREFP 3 C00265 BC00265  +REFP EC00265
CALL JOB:SEARCH-R1-S13D
SET P051 P006
SFTON3D P051
SMOVL C00266 BC00266 V=166.7  +MOVJ EC00266
SREFP 3 C00267 BC00267  +REFP EC00267
CALL JOB:SEARCH-R1-S13D
SET P051 P006
SFTON3D P051
SMOVL C00268 BC00268 V=166.7  +MOVJ EC00268
MOVL C00269 BC00269 V=333.3  +MOVJ EC00269 VJ=100.00
'EndPath S3365
'Path S3366
SFTOF3D
MOVL C00270 BC00270 V=800.0  +MOVJ EC00270 VJ=100.00
SMOVL C00271 BC00271 V=166.7  +MOVJ EC00271
SREFP 3 C00272 BC00272  +REFP EC00272
CALL JOB:SEARCH-R1-S13D
SET P052 P006
SFTON3D P052
SMOVL C00273 BC00273 V=166.7  +MOVJ EC00273
SREFP 3 C00274 BC00274  +REFP EC00274
CALL JOB:SEARCH-R1-S13D
SET P052 P006
SFTON3D P052
SMOVL C00275 BC00275 V=166.7  +MOVJ EC00275
'EndPath S3366
'Path S3367
SFTOF3D
MOVL C00276 BC00276 V=800.0  +MOVJ EC00276 VJ=100.00
SMOVL C00277 BC00277 V=166.7  +MOVJ EC00277
SREFP 3 C00278 BC00278  +REFP EC00278
CALL JOB:SEARCH-R1-S13D
SET P053 P006
SFTON3D P053
SMOVL C00279 BC00279 V=166.7  +MOVJ EC00279
SREFP 3 C00280 BC00280  +REFP EC00280
CALL JOB:SEARCH-R1-S13D
SET P053 P006
SFTON3D P053
SMOVL C00281 BC00281 V=166.7  +MOVJ EC00281
SFTOF3D
MOVL C00282 BC00282 V=333.3  +MOVJ EC00282 VJ=100.00
'EndPath S3367
'
'Path W3331
SFTOF3D
SFTON3D P052
SMOVL C00283 BC00283 V=150.0 PL=0  +MOVJ EC00283
ARCON
SFTON3D P053
SMOVL C00284 BC00284 V=9.2  +MOVJ EC00284
ARCOF
SMOVL C00285 BC00285 V=800.0  +MOVJ EC00285
SMOVL C00286 BC00286 V=1000.0  +MOVJ EC00286
SFTOF3D
'EndPath W3331
MOVJ C00287 BC00287 VJ=100.00  +MOVJ EC00287 VJ=100.00
'
'Path W3335
SFTOF3D
SFTON3D P051
SMOVL C00288 BC00288 V=800.0  +MOVJ EC00288
SMOVL C00289 BC00289 V=150.0 PL=0  +MOVJ EC00289
ARCON
SFTON3D P050
SMOVL C00290 BC00290 V=9.2  +MOVJ EC00290
ARCOF
SMOVL C00291 BC00291 V=416.7  +MOVJ EC00291
SMOVL C00292 BC00292 V=500.0  +MOVJ EC00292
SFTOF3D
'EndPath W3335
'
'Path W3326
SFTOF3D
SFTON3D P047
MOVJ C00293 BC00293 VJ=100.00  +MOVJ EC00293 VJ=100.00
SMOVL C00294 BC00294 V=800.0  +MOVJ EC00294
SMOVL C00295 BC00295 V=150.0 PL=0  +MOVJ EC00295
MACRO1 MJ#(0) ARGF9
ARCON
SMOVL C00296 BC00296 V=11.7  +MOVJ EC00296
ARCOF
SMOVL C00297 BC00297 V=800.0  +MOVJ EC00297
SMOVL C00298 BC00298 V=500.0  +MOVJ EC00298
SFTOF3D
'EndPath W3326
'Path W3327
SFTOF3D
SFTON3D P048
MOVJ C00299 BC00299 VJ=100.00  +MOVJ EC00299 VJ=100.00
SMOVL C00300 BC00300 V=800.0  +MOVJ EC00300
SMOVL C00301 BC00301 V=150.0 PL=0  +MOVJ EC00301
ARCON
SMOVL C00302 BC00302 V=11.7  +MOVJ EC00302
ARCOF
SMOVL C00303 BC00303 V=800.0  +MOVJ EC00303
SMOVL C00304 BC00304 V=333.3  +MOVJ EC00304
'Path W3328
SFTOF3D
SFTON3D P045
MOVJ C00305 BC00305 VJ=100.00  +MOVJ EC00305 VJ=100.00
SMOVL C00306 BC00306 V=800.0  +MOVJ EC00306
SMOVL C00307 BC00307 V=150.0 PL=0  +MOVJ EC00307
ARCON
SMOVL C00308 BC00308 V=11.7  +MOVJ EC00308
ARCOF
SMOVL C00309 BC00309 V=800.0  +MOVJ EC00309
SFTOF3D
'EndPath W3324
'Path W3325
SFTOF3D
SFTON3D P046
MOVJ C00310 BC00310 VJ=20.00  +MOVJ EC00310 VJ=20.00
MOVJ C00311 BC00311 VJ=20.00  +MOVJ EC00311 VJ=100.00
SMOVL C00312 BC00312 V=800.0  +MOVJ EC00312
SMOVL C00313 BC00313 V=150.0 PL=0  +MOVJ EC00313
ARCON
SMOVL C00314 BC00314 V=11.7  +MOVJ EC00314
ARCOF
SMOVL C00315 BC00315 V=500.0  +MOVJ EC00315
SFTOF3D
'EndPath W3325
'
'
'Path W3320
SFTOF3D
SFTON3D P041
MOVJ C00316 BC00316 VJ=100.00  +MOVJ EC00316 VJ=100.00
SMOVL C00317 BC00317 V=800.0  +MOVJ EC00317
SMOVL C00318 BC00318 V=166.7 PL=0  +MOVJ EC00318
ARCON
SMOVL C00319 BC00319 V=11.7  +MOVJ EC00319
ARCOF
SMOVL C00320 BC00320 V=333.3  +MOVJ EC00320
SFTOF3D
'EndPath W3320
'Path W3321
SFTOF3D
SFTON3D P042
MOVJ C00321 BC00321 VJ=20.00  +MOVJ EC00321 VJ=20.00
MOVJ C00322 BC00322 VJ=100.00  +MOVJ EC00322 VJ=100.00
SMOVL C00323 BC00323 V=800.0  +MOVJ EC00323
SMOVL C00324 BC00324 V=166.7 PL=0  +MOVJ EC00324
ARCON
SMOVL C00325 BC00325 V=11.7  +MOVJ EC00325
ARCOF
SMOVL C00326 BC00326 V=800.0  +MOVJ EC00326
SFTOF3D
MOVJ C00327 BC00327 VJ=20.00  +MOVJ EC00327 VJ=100.00
MOVJ C00328 BC00328 VJ=20.00  +MOVJ EC00328 VJ=100.00
MOVJ C00329 BC00329 VJ=20.00  +MOVJ EC00329 VJ=100.00
MOVJ C00330 BC00330 VJ=20.00  +MOVJ EC00330 VJ=100.00
MOVJ C00331 BC00331 VJ=20.00  +MOVJ EC00331 VJ=20.00
MOVJ C00332 BC00332 VJ=20.00  +MOVJ EC00332 VJ=20.00
MOVJ C00333 BC00333 VJ=20.00  +MOVJ EC00333 VJ=100.00
MOVJ C00334 BC00334 VJ=20.00  +MOVJ EC00334 VJ=20.00
CALL JOB:CLEAN-R1_KM_NEW
MOVJ C00335 BC00335 VJ=100.00  +MOVJ EC00335 VJ=100.00
'
'Path S3355
SFTOF3D
MOVJ C00336 BC00336 VJ=100.00  +MOVJ EC00336 VJ=100.00
MOVL C00337 BC00337 V=800.0  +MOVJ EC00337 VJ=100.00
MOVL C00338 BC00338 V=800.0  +MOVJ EC00338 VJ=100.00
SMOVL C00339 BC00339 V=166.7  +MOVJ EC00339
SREFP 3 C00340 BC00340  +REFP EC00340
CALL JOB:SEARCH-R1-S13D
SET P041 P006
SFTON3D P041
SMOVL C00341 BC00341 V=166.7  +MOVJ EC00341
SREFP 3 C00342 BC00342  +REFP EC00342
CALL JOB:SEARCH-R1-S13D
SET P041 P006
SFTON3D P041
SMOVL C00343 BC00343 V=166.7  +MOVJ EC00343
MOVL C00344 BC00344 V=1000.0  +MOVJ EC00344 VJ=100.00
'EndPath S3355
'Path S3356
SFTOF3D
MOVJ C00345 BC00345 VJ=100.00  +MOVJ EC00345 VJ=100.00
MOVL C00346 BC00346 V=800.0  +MOVJ EC00346 VJ=100.00
SMOVL C00347 BC00347 V=166.7  +MOVJ EC00347
SREFP 3 C00348 BC00348  +REFP EC00348
CALL JOB:SEARCH-R1-S13D
SET P042 P006
SFTON3D P042
SMOVL C00349 BC00349 V=166.7  +MOVJ EC00349
SREFP 3 C00350 BC00350  +REFP EC00350
CALL JOB:SEARCH-R1-S13D
SET P042 P006
SFTON3D P042
SMOVL C00351 BC00351 V=166.7  +MOVJ EC00351
MOVL C00352 BC00352 V=1000.0  +MOVJ EC00352 VJ=100.00
'EndPath S3356
SFTOF3D
MOVJ C00353 BC00353 VJ=100.00  +MOVJ EC00353 VJ=100.00
SFTOF3D
MOVJ C00354 BC00354 VJ=100.00  +MOVJ EC00354 VJ=100.00
MOVL C00355 BC00355 V=800.0  +MOVJ EC00355 VJ=100.00
SMOVL C00356 BC00356 V=166.7  +MOVJ EC00356
SREFP 3 C00357 BC00357  +REFP EC00357
CALL JOB:SEARCH-R1-S13D
SET P045 P006
SFTON3D P045
SMOVL C00358 BC00358 V=166.7  +MOVJ EC00358
SREFP 3 C00359 BC00359  +REFP EC00359
CALL JOB:SEARCH-R1-S13D
SET P045 P006
SFTON3D P045
SMOVL C00360 BC00360 V=166.7  +MOVJ EC00360
MOVL C00361 BC00361 V=1000.0  +MOVJ EC00361 VJ=100.00
'EndPath S3359
'Path S3360
SFTOF3D
MOVJ C00362 BC00362 VJ=100.00  +MOVJ EC00362 VJ=100.00
MOVL C00363 BC00363 V=800.0  +MOVJ EC00363 VJ=100.00
SMOVL C00364 BC00364 V=166.7  +MOVJ EC00364
SREFP 3 C00365 BC00365  +REFP EC00365
CALL JOB:SEARCH-R1-S13D
SET P046 P006
SFTON3D P046
SMOVL C00366 BC00366 V=166.7  +MOVJ EC00366
SREFP 3 C00367 BC00367  +REFP EC00367
CALL JOB:SEARCH-R1-S13D
SET P046 P006
SFTON3D P046
SMOVL C00368 BC00368 V=166.7  +MOVJ EC00368
MOVL C00369 BC00369 V=1000.0  +MOVJ EC00369 VJ=100.00
'EndPath S3360
MOVJ C00370 BC00370 VJ=100.00  +MOVJ EC00370 VJ=100.00
'Path S3361
SFTOF3D
MOVJ C00371 BC00371 VJ=100.00  +MOVJ EC00371 VJ=100.00
MOVL C00372 BC00372 V=800.0  +MOVJ EC00372 VJ=100.00
SMOVL C00373 BC00373 V=166.7  +MOVJ EC00373
SREFP 3 C00374 BC00374  +REFP EC00374
CALL JOB:SEARCH-R1-S13D
SET P047 P006
SFTON3D P047
SMOVL C00375 BC00375 V=166.7  +MOVJ EC00375
SREFP 3 C00376 BC00376  +REFP EC00376
CALL JOB:SEARCH-R1-S13D
SET P047 P006
SFTON3D P047
SMOVL C00377 BC00377 V=166.7  +MOVJ EC00377
MOVL C00378 BC00378 V=1000.0  +MOVJ EC00378 VJ=100.00
'EndPath S3361
'Path S3362
SFTOF3D
MOVJ C00379 BC00379 VJ=100.00  +MOVJ EC00379 VJ=100.00
MOVL C00380 BC00380 V=800.0  +MOVJ EC00380 VJ=100.00
SMOVL C00381 BC00381 V=166.7  +MOVJ EC00381
SREFP 3 C00382 BC00382  +REFP EC00382
CALL JOB:SEARCH-R1-S13D
SET P048 P006
SFTON3D P048
SMOVL C00383 BC00383 V=166.7  +MOVJ EC00383
SREFP 3 C00384 BC00384  +REFP EC00384
CALL JOB:SEARCH-R1-S13D
SET P048 P006
SFTON3D P048
SMOVL C00385 BC00385 V=166.7  +MOVJ EC00385
MOVL C00386 BC00386 V=1000.0  +MOVJ EC00386 VJ=100.00
'EndPath S3362
'Path S3363
SFTOF3D
MOVJ C00387 BC00387 VJ=100.00  +MOVJ EC00387 VJ=100.00
MOVL C00388 BC00388 V=333.3  +MOVJ EC00388 VJ=100.00
SMOVL C00389 BC00389 V=166.7  +MOVJ EC00389
SREFP 3 C00390 BC00390  +REFP EC00390
CALL JOB:SEARCH-R1-S13D
SET P050 P006
SFTON3D P050
SMOVL C00391 BC00391 V=166.7  +MOVJ EC00391
SREFP 3 C00392 BC00392  +REFP EC00392
CALL JOB:SEARCH-R1-S13D
SET P050 P006
SFTON3D P050
SMOVL C00393 BC00393 V=166.7  +MOVJ EC00393
'EndPath S3364
'Path S3365
SFTOF3D
MOVJ C00394 BC00394 VJ=100.00  +MOVJ EC00394 VJ=100.00
MOVL C00395 BC00395 V=800.0  +MOVJ EC00395 VJ=100.00
SMOVL C00396 BC00396 V=166.7  +MOVJ EC00396
SREFP 3 C00397 BC00397  +REFP EC00397
CALL JOB:SEARCH-R1-S13D
SET P051 P006
SFTON3D P051
SMOVL C00398 BC00398 V=166.7  +MOVJ EC00398
SREFP 3 C00399 BC00399  +REFP EC00399
CALL JOB:SEARCH-R1-S13D
SET P051 P006
SFTON3D P051
SMOVL C00400 BC00400 V=166.7  +MOVJ EC00400
MOVL C00401 BC00401 V=1000.0  +MOVJ EC00401 VJ=100.00
'EndPath S3365
MOVJ C00402 BC00402 VJ=100.00  +MOVJ EC00402 VJ=100.00
'Path S3366
SFTOF3D
MOVL C00403 BC00403 V=800.0  +MOVJ EC00403 VJ=100.00
SMOVL C00404 BC00404 V=166.7  +MOVJ EC00404
SREFP 3 C00405 BC00405  +REFP EC00405
CALL JOB:SEARCH-R1-S13D
SET P052 P006
SFTON3D P052
SMOVL C00406 BC00406 V=166.7  +MOVJ EC00406
SREFP 3 C00407 BC00407  +REFP EC00407
CALL JOB:SEARCH-R1-S13D
SET P052 P006
SFTON3D P052
SMOVL C00408 BC00408 V=166.7  +MOVJ EC00408
MOVL C00409 BC00409 V=1000.0  +MOVJ EC00409 VJ=100.00
'EndPath S3366
'Path S3367
SFTOF3D
SMOVL C00410 BC00410 V=166.7  +MOVJ EC00410
SREFP 3 C00411 BC00411  +REFP EC00411
CALL JOB:SEARCH-R1-S13D
SET P053 P006
SFTON3D P053
SMOVL C00412 BC00412 V=166.7  +MOVJ EC00412
SREFP 3 C00413 BC00413  +REFP EC00413
CALL JOB:SEARCH-R1-S13D
SET P053 P006
SFTON3D P053
SMOVL C00414 BC00414 V=166.7  +MOVJ EC00414
SFTOF3D
'EndPath S3367
'
'Path W3331
SFTOF3D
SFTON3D P053
SMOVL C00415 BC00415 V=150.0 PL=0  +MOVJ EC00415
ARCON
SFTON3D P052
SMOVL C00416 BC00416 V=9.2  +MOVJ EC00416
ARCOF
SMOVL C00417 BC00417 V=800.0  +MOVJ EC00417
SMOVL C00418 BC00418 V=1000.0  +MOVJ EC00418
SFTOF3D
'EndPath W3331
'
'Path W3335
SFTOF3D
SFTON3D P051
SMOVL C00419 BC00419 V=800.0  +MOVJ EC00419
SMOVL C00420 BC00420 V=150.0 PL=0  +MOVJ EC00420
ARCON
SFTON3D P050
SMOVL C00421 BC00421 V=10.0  +MOVJ EC00421
ARCOF
SMOVL C00422 BC00422 V=800.0  +MOVJ EC00422
SMOVL C00423 BC00423 V=1000.0  +MOVJ EC00423
SFTOF3D
'EndPath W3335
'
'Path W3326
SFTOF3D
SFTON3D P047
MOVJ C00424 BC00424 VJ=100.00  +MOVJ EC00424 VJ=100.00
SMOVL C00425 BC00425 V=800.0  +MOVJ EC00425
SMOVL C00426 BC00426 V=150.0 PL=0  +MOVJ EC00426
MACRO1 MJ#(0) ARGF9
ARCON
SMOVL C00427 BC00427 V=11.7  +MOVJ EC00427
ARCOF
SMOVL C00428 BC00428 V=800.0  +MOVJ EC00428
SMOVL C00429 BC00429 V=1000.0  +MOVJ EC00429
SFTOF3D
'EndPath W3326
'Path W3327
SFTOF3D
SFTON3D P048
MOVJ C00430 BC00430 VJ=100.00  +MOVJ EC00430 VJ=100.00
SMOVL C00431 BC00431 V=800.0  +MOVJ EC00431
SMOVL C00432 BC00432 V=150.0 PL=0  +MOVJ EC00432
ARCON
SMOVL C00433 BC00433 V=11.7  +MOVJ EC00433
ARCOF
SMOVL C00434 BC00434 V=800.0  +MOVJ EC00434
SMOVL C00435 BC00435 V=1000.0  +MOVJ EC00435
SFTOF3D
'Path W3324
SFTOF3D
SFTON3D P045
MOVJ C00436 BC00436 VJ=100.00  +MOVJ EC00436 VJ=100.00
SMOVL C00437 BC00437 V=800.0  +MOVJ EC00437
SMOVL C00438 BC00438 V=150.0 PL=0  +MOVJ EC00438
ARCON
SMOVL C00439 BC00439 V=11.7  +MOVJ EC00439
ARCOF
SMOVL C00440 BC00440 V=800.0  +MOVJ EC00440
SMOVL C00441 BC00441 V=500.0  +MOVJ EC00441
SFTOF3D
'EndPath W3324
'Path W3325
SFTOF3D
SFTON3D P046
MOVJ C00442 BC00442 VJ=100.00  +MOVJ EC00442 VJ=100.00
SMOVL C00443 BC00443 V=800.0  +MOVJ EC00443
SMOVL C00444 BC00444 V=150.0 PL=0  +MOVJ EC00444
ARCON
SMOVL C00445 BC00445 V=11.7  +MOVJ EC00445
ARCOF
SMOVL C00446 BC00446 V=800.0  +MOVJ EC00446
SMOVL C00447 BC00447 V=1000.0  +MOVJ EC00447
SFTOF3D
'EndPath W3325
MOVJ C00448 BC00448 VJ=100.00  +MOVJ EC00448 VJ=100.00
'
'
'Path W3320
SFTOF3D
SFTON3D P041
MOVJ C00449 BC00449 VJ=100.00  +MOVJ EC00449 VJ=100.00
SMOVL C00450 BC00450 V=800.0  +MOVJ EC00450
SMOVL C00451 BC00451 V=166.7 PL=0  +MOVJ EC00451
ARCON
SMOVL C00452 BC00452 V=11.7  +MOVJ EC00452
ARCOF
SMOVL C00453 BC00453 V=800.0  +MOVJ EC00453
SMOVL C00454 BC00454 V=1000.0  +MOVJ EC00454
SFTOF3D
'EndPath W3320
'Path W3321
SFTOF3D
SFTON3D P042
MOVJ C00455 BC00455 VJ=100.00  +MOVJ EC00455 VJ=100.00
SMOVL C00456 BC00456 V=800.0  +MOVJ EC00456
SMOVL C00457 BC00457 V=166.7 PL=0  +MOVJ EC00457
ARCON
SMOVL C00458 BC00458 V=11.7  +MOVJ EC00458
ARCOF
SMOVL C00459 BC00459 V=800.0  +MOVJ EC00459
SMOVL C00460 BC00460 V=1000.0  +MOVJ EC00460
SFTOF3D
MOVJ C00461 BC00461 VJ=20.00  +MOVJ EC00461 VJ=100.00
MOVJ C00462 BC00462 VJ=20.00  +MOVJ EC00462 VJ=20.00
MOVJ C00463 BC00463 VJ=15.00  +MOVJ EC00463 VJ=100.00
MOVJ C00464 BC00464 VJ=15.00  +MOVJ EC00464 VJ=100.00
END
